LIN {X 107.589,Y -46.162,Z -55.457,A -90.000,B 90.000,C 0.000} C_DIS
LIN {X 107.509,Y -46.153,Z -55.761,A -90.000,B 90.000,C 0.000} C_DIS
LIN {X 107.348,Y -46.129,Z -56.352,A -90.000,B 90.000,C 0.000} C_DIS
LIN {X 107.212,Y -46.114,Z -56.832,A -90.000,B 90.000,C 0.000} C_DIS
LIN {X 107.081,Y -46.091,Z -57.259,A -90.000,B 90.000,C 0.000} C_DIS
LIN {X 106.960,Y -46.087,Z -57.631,A -90.000,B 90.000,C 0.000} C_DIS
LIN {X 106.873,Y -46.081,Z -57.884,A -90.000,B 90.000,C 0.000} C_DIS
LIN {X 106.583,Y -46.065,Z -58.706,A -90.000,B 90.000,C 0.000} C_DIS
LIN {X 106.300,Y -46.057,Z -59.526,A -90.000,B 90.000,C 0.000} C_DIS
LIN {X 106.266,Y -46.058,Z -59.619,A -90.000,B 90.000,C 0.000} C_DIS
LIN {X 106.210,Y -46.061,Z -59.764,A -90.000,B 90.000,C 0.000} C_DIS
LIN {X 105.890,Y -46.060,Z -60.546,A -90.000,B 90.000,C 0.000} C_DIS
LIN {X 105.587,Y -46.066,Z -61.296,A -90.000,B 90.000,C 0.000} C_DIS
LIN {X 105.326,Y -46.072,Z -61.938,A -90.000,B 90.000,C 0.000} C_DIS
LIN {X 105.166,Y -46.078,Z -62.307,A -90.000,B 90.000,C 0.000} C_DIS
LIN {X 104.885,Y -46.086,Z -62.880,A -90.000,B 90.000,C 0.000} C_DIS
LIN {X 104.370,Y -46.110,Z -63.945,A -90.000,B 90.000,C 0.000} C_DIS
LIN {X 104.116,Y -46.117,Z -64.480,A -90.000,B 90.000,C 0.000} C_DIS
LIN {X 104.061,Y -46.121,Z -64.587,A -90.000,B 90.000,C 0.000} C_DIS
LIN {X 103.858,Y -46.124,Z -64.941,A -90.000,B 90.000,C 0.000} C_DIS
LIN {X 103.565,Y -46.141,Z -65.429,A -90.000,B 90.000,C 0.000} C_DIS
LIN {X 102.922,Y -46.183,Z -66.506,A -90.000,B 90.000,C 0.000} C_DIS
LIN {X 102.789,Y -46.189,Z -66.734,A -90.000,B 90.000,C 0.000} C_DIS
LIN {X 102.578,Y -46.188,Z -67.081,A -90.000,B 90.000,C 0.000} C_DIS
LIN {X 102.463,Y -46.188,Z -67.247,A -90.000,B 90.000,C 0.000} C_DIS
LIN {X 102.227,Y -46.200,Z -67.560,A -90.000,B 90.000,C 0.000} C_DIS
LIN {X 101.675,Y -46.239,Z -68.268,A -90.000,B 90.000,C 0.000} C_DIS
LIN {X 101.476,Y -46.259,Z -68.509,A -90.000,B 90.000,C 0.000} C_DIS
LIN {X 101.020,Y -46.294,Z -69.044,A -90.000,B 90.000,C 0.000} C_DIS
LIN {X 100.781,Y -46.305,Z -69.318,A -90.000,B 90.000,C 0.000} C_DIS
LIN {X 100.500,Y -46.311,Z -69.634,A -90.000,B 90.000,C 0.000} C_DIS
LIN {X 100.413,Y -46.315,Z -69.726,A -90.000,B 90.000,C 0.000} C_DIS
LIN {X 100.368,Y -46.319,Z -69.770,A -90.000,B 90.000,C 0.000} C_DIS
LIN {X 100.015,Y -46.339,Z -70.076,A -90.000,B 90.000,C 0.000} C_DIS
LIN {X 99.523,Y -46.377,Z -70.476,A -90.000,B 90.000,C 0.000} C_DIS
LIN {X 98.816,Y -46.424,Z -71.045,A -90.000,B 90.000,C 0.000} C_DIS
LIN {X 98.553,Y -46.429,Z -71.249,A -90.000,B 90.000,C 0.000} C_DIS
LIN {X 97.950,Y -46.427,Z -71.707,A -90.000,B 90.000,C 0.000} C_DIS
LIN {X 97.860,Y -46.428,Z -71.773,A -90.000,B 90.000,C 0.000} C_DIS
LIN {X 97.743,Y -46.434,Z -71.848,A -90.000,B 90.000,C 0.000} C_DIS
LIN {X 97.472,Y -46.450,Z -72.014,A -90.000,B 90.000,C 0.000} C_DIS
LIN {X 97.222,Y -46.468,Z -72.161,A -90.000,B 90.000,C 0.000} C_DIS
LIN {X 97.080,Y -46.480,Z -72.238,A -90.000,B 90.000,C 0.000} C_DIS
LIN {X 96.822,Y -46.489,Z -72.366,A -90.000,B 90.000,C 0.000} C_DIS
LIN {X 96.112,Y -46.501,Z -72.711,A -90.000,B 90.000,C 0.000} C_DIS
LIN {X 95.963,Y -46.506,Z -72.774,A -90.000,B 90.000,C 0.000} C_DIS
LIN {X 95.665,Y -46.507,Z -72.890,A -90.000,B 90.000,C 0.000} C_DIS
LIN {X 95.513,Y -46.511,Z -72.938,A -90.000,B 90.000,C 0.000} C_DIS
LIN {X 94.694,Y -46.547,Z -73.167,A -90.000,B 90.000,C 0.000} C_DIS
LIN {X 94.626,Y -46.549,Z -73.189,A -90.000,B 90.000,C 0.000} C_DIS
LIN {X 94.421,Y -46.549,Z -73.252,A -90.000,B 90.000,C 0.000} C_DIS
LIN {X 94.032,Y -46.560,Z -73.343,A -90.000,B 90.000,C 0.000} C_DIS
LIN {X 93.943,Y -46.563,Z -73.362,A -90.000,B 90.000,C 0.000} C_DIS
LIN {X 93.880,Y -46.566,Z -73.372,A -90.000,B 90.000,C 0.000} C_DIS
LIN {X 93.755,Y -46.574,Z -73.389,A -90.000,B 90.000,C 0.000} C_DIS
LIN {X 93.477,Y -46.578,Z -73.425,A -90.000,B 90.000,C 0.000} C_DIS
LIN {X 92.687,Y -46.571,Z -73.521,A -90.000,B 90.000,C 0.000} C_DIS
LIN {X 92.591,Y -46.573,Z -73.532,A -90.000,B 90.000,C 0.000} C_DIS
LIN {X 92.407,Y -46.579,Z -73.545,A -90.000,B 90.000,C 0.000} C_DIS
LIN {X 92.089,Y -46.581,Z -73.541,A -90.000,B 90.000,C 0.000} C_DIS
LIN {X 92.022,Y -46.582,Z -73.539,A -90.000,B 90.000,C 0.000} C_DIS
LIN {X 91.526,Y -46.592,Z -73.502,A -90.000,B 90.000,C 0.000} C_DIS
LIN {X 91.111,Y -46.595,Z -73.489,A -90.000,B 90.000,C 0.000} C_DIS
LIN {X 91.023,Y -46.591,Z -73.484,A -90.000,B 90.000,C 0.000} C_DIS
LIN {X 90.905,Y -46.587,Z -73.475,A -90.000,B 90.000,C 0.000} C_DIS
LIN {X 90.779,Y -46.586,Z -73.457,A -90.000,B 90.000,C 0.000} C_DIS
LIN {X 90.544,Y -46.586,Z -73.417,A -90.000,B 90.000,C 0.000} C_DIS
LIN {X 90.416,Y -46.588,Z -73.388,A -90.000,B 90.000,C 0.000} C_DIS
LIN {X 90.003,Y -46.595,Z -73.288,A -90.000,B 90.000,C 0.000} C_DIS
LIN {X 89.846,Y -46.594,Z -73.260,A -90.000,B 90.000,C 0.000} C_DIS
LIN {X 89.559,Y -46.578,Z -73.201,A -90.000,B 90.000,C 0.000} C_DIS
LIN {X 89.440,Y -46.573,Z -73.172,A -90.000,B 90.000,C 0.000} C_DIS
LIN {X 89.132,Y -46.563,Z -73.088,A -90.000,B 90.000,C 0.000} C_DIS
LIN {X 89.029,Y -46.561,Z -73.057,A -90.000,B 90.000,C 0.000} C_DIS
LIN {X 88.840,Y -46.562,Z -72.987,A -90.000,B 90.000,C 0.000} C_DIS
LIN {X 88.626,Y -46.563,Z -72.902,A -90.000,B 90.000,C 0.000} C_DIS
LIN {X 88.200,Y -46.542,Z -72.723,A -90.000,B 90.000,C 0.000} C_DIS
LIN {X 87.848,Y -46.530,Z -72.563,A -90.000,B 90.000,C 0.000} C_DIS
LIN {X 87.511,Y -46.517,Z -72.389,A -90.000,B 90.000,C 0.000} C_DIS
LIN {X 87.327,Y -46.505,Z -72.292,A -90.000,B 90.000,C 0.000} C_DIS
LIN {X 87.280,Y -46.500,Z -72.274,A -90.000,B 90.000,C 0.000} C_DIS
LIN {X 87.174,Y -46.490,Z -72.230,A -90.000,B 90.000,C 0.000} C_DIS
LIN {X 87.006,Y -46.476,Z -72.150,A -90.000,B 90.000,C 0.000} C_DIS
LIN {X 86.828,Y -46.472,Z -72.071,A -90.000,B 90.000,C 0.000} C_DIS
LIN {X 86.767,Y -46.472,Z -72.041,A -90.000,B 90.000,C 0.000} C_DIS
LIN {X 86.689,Y -46.469,Z -71.999,A -90.000,B 90.000,C 0.000} C_DIS
LIN {X 86.578,Y -46.468,Z -71.932,A -90.000,B 90.000,C 0.000} C_DIS
LIN {X 86.493,Y -46.468,Z -71.878,A -90.000,B 90.000,C 0.000} C_DIS
LIN {X 86.279,Y -46.453,Z -71.731,A -90.000,B 90.000,C 0.000} C_DIS
LIN {X 85.850,Y -46.419,Z -71.423,A -90.000,B 90.000,C 0.000} C_DIS
LIN {X 85.760,Y -46.408,Z -71.369,A -90.000,B 90.000,C 0.000} C_DIS
LIN {X 85.585,Y -46.403,Z -71.258,A -90.000,B 90.000,C 0.000} C_DIS
LIN {X 85.416,Y -46.390,Z -71.143,A -90.000,B 90.000,C 0.000} C_DIS
LIN {X 85.343,Y -46.385,Z -71.090,A -90.000,B 90.000,C 0.000} C_DIS
LIN {X 85.266,Y -46.378,Z -71.028,A -90.000,B 90.000,C 0.000} C_DIS
LIN {X 85.091,Y -46.365,Z -70.871,A -90.000,B 90.000,C 0.000} C_DIS
LIN {X 85.014,Y -46.355,Z -70.797,A -90.000,B 90.000,C 0.000} C_DIS
LIN {X 84.936,Y -46.346,Z -70.718,A -90.000,B 90.000,C 0.000} C_DIS
LIN {X 84.756,Y -46.327,Z -70.529,A -90.000,B 90.000,C 0.000} C_DIS
LIN {X 84.658,Y -46.327,Z -70.434,A -90.000,B 90.000,C 0.000} C_DIS
LIN {X 84.355,Y -46.303,Z -70.183,A -90.000,B 90.000,C 0.000} C_DIS
LIN {X 84.253,Y -46.288,Z -70.085,A -90.000,B 90.000,C 0.000} C_DIS
LIN {X 84.127,Y -46.274,Z -69.947,A -90.000,B 90.000,C 0.000} C_DIS
LIN {X 83.956,Y -46.242,Z -69.742,A -90.000,B 90.000,C 0.000} C_DIS
LIN {X 83.874,Y -46.226,Z -69.634,A -90.000,B 90.000,C 0.000} C_DIS
LIN {X 83.782,Y -46.213,Z -69.499,A -90.000,B 90.000,C 0.000} C_DIS
LIN {X 83.711,Y -46.202,Z -69.388,A -90.000,B 90.000,C 0.000} C_DIS
LIN {X 83.619,Y -46.198,Z -69.257,A -90.000,B 90.000,C 0.000} C_DIS
LIN {X 83.569,Y -46.197,Z -69.184,A -90.000,B 90.000,C 0.000} C_DIS
LIN {X 83.433,Y -46.199,Z -68.968,A -90.000,B 90.000,C 0.000} C_DIS
LIN {X 83.314,Y -46.181,Z -68.793,A -90.000,B 90.000,C 0.000} C_DIS
LIN {X 83.245,Y -46.172,Z -68.688,A -90.000,B 90.000,C 0.000} C_DIS
LIN {X 83.110,Y -46.136,Z -68.456,A -90.000,B 90.000,C 0.000} C_DIS
LIN {X 82.973,Y -46.109,Z -68.193,A -90.000,B 90.000,C 0.000} C_DIS
LIN {X 82.834,Y -46.065,Z -67.863,A -90.000,B 90.000,C 0.000} C_DIS
LIN {X 82.812,Y -46.055,Z -67.802,A -90.000,B 90.000,C 0.000} C_DIS
LIN {X 82.777,Y -46.044,Z -67.715,A -90.000,B 90.000,C 0.000} C_DIS
LIN {X 82.723,Y -46.031,Z -67.563,A -90.000,B 90.000,C 0.000} C_DIS
LIN {X 82.697,Y -46.027,Z -67.483,A -90.000,B 90.000,C 0.000} C_DIS
LIN {X 82.592,Y -46.003,Z -67.135,A -90.000,B 90.000,C 0.000} C_DIS
LIN {X 82.505,Y -45.973,Z -66.741,A -90.000,B 90.000,C 0.000} C_DIS
LIN {X 82.442,Y -45.940,Z -66.413,A -90.000,B 90.000,C 0.000} C_DIS
LIN {X 82.413,Y -45.927,Z -66.257,A -90.000,B 90.000,C 0.000} C_DIS
LIN {X 82.375,Y -45.874,Z -65.905,A -90.000,B 90.000,C 0.000} C_DIS
LIN {X 82.362,Y -45.850,Z -65.730,A -90.000,B 90.000,C 0.000} C_DIS
LIN {X 82.347,Y -45.818,Z -65.409,A -90.000,B 90.000,C 0.000} C_DIS
LIN {X 82.364,Y -45.773,Z -65.034,A -90.000,B 90.000,C 0.000} C_DIS
LIN {X 82.401,Y -45.734,Z -64.565,A -90.000,B 90.000,C 0.000} C_DIS
LIN {X 82.410,Y -45.729,Z -64.470,A -90.000,B 90.000,C 0.000} C_DIS
LIN {X 82.479,Y -45.709,Z -63.856,A -90.000,B 90.000,C 0.000} C_DIS
LIN {X 82.501,Y -45.701,Z -63.740,A -90.000,B 90.000,C 0.000} C_DIS
LIN {X 82.576,Y -45.681,Z -63.378,A -90.000,B 90.000,C 0.000} C_DIS
LIN {X 82.598,Y -45.674,Z -63.301,A -90.000,B 90.000,C 0.000} C_DIS
LIN {X 82.709,Y -45.640,Z -62.934,A -90.000,B 90.000,C 0.000} C_DIS
LIN {X 82.820,Y -45.612,Z -62.579,A -90.000,B 90.000,C 0.000} C_DIS
LIN {X 83.043,Y -45.545,Z -62.002,A -90.000,B 90.000,C 0.000} C_DIS
LIN {X 83.069,Y -45.539,Z -61.937,A -90.000,B 90.000,C 0.000} C_DIS
LIN {X 83.136,Y -45.526,Z -61.772,A -90.000,B 90.000,C 0.000} C_DIS
LIN {X 83.311,Y -45.490,Z -61.398,A -90.000,B 90.000,C 0.000} C_DIS
LIN {X 83.482,Y -45.470,Z -61.064,A -90.000,B 90.000,C 0.000} C_DIS
LIN {X 83.601,Y -45.459,Z -60.837,A -90.000,B 90.000,C 0.000} C_DIS
LIN {X 83.737,Y -45.451,Z -60.585,A -90.000,B 90.000,C 0.000} C_DIS
LIN {X 83.897,Y -45.437,Z -60.318,A -90.000,B 90.000,C 0.000} C_DIS
LIN {X 84.064,Y -45.422,Z -60.072,A -90.000,B 90.000,C 0.000} C_DIS
LIN {X 84.175,Y -45.411,Z -59.915,A -90.000,B 90.000,C 0.000} C_DIS
LIN {X 84.538,Y -45.384,Z -59.413,A -90.000,B 90.000,C 0.000} C_DIS
LIN {X 84.832,Y -45.368,Z -59.006,A -90.000,B 90.000,C 0.000} C_DIS
LIN {X 85.043,Y -45.360,Z -58.718,A -90.000,B 90.000,C 0.000} C_DIS
LIN {X 85.401,Y -45.345,Z -58.270,A -90.000,B 90.000,C 0.000} C_DIS
LIN {X 85.618,Y -45.344,Z -57.999,A -90.000,B 90.000,C 0.000} C_DIS
LIN {X 85.618,Y -60.000,Z -57.999,A -90.000,B 90.000,C 0.000} C_DIS
LIN {X 100.781,Y -60.000,Z -71.645,A -90.000,B 90.000,C 0.000} C_DIS
LIN {X 100.781,Y -45.308,Z -71.645,A -90.000,B 90.000,C 0.000} C_DIS
LIN {X 100.498,Y -45.352,Z -71.891,A -90.000,B 90.000,C 0.000} C_DIS
LIN {X 99.019,Y -45.480,Z -73.108,A -90.000,B 90.000,C 0.000} C_DIS
LIN {X 98.875,Y -45.494,Z -73.221,A -90.000,B 90.000,C 0.000} C_DIS
LIN {X 98.794,Y -45.505,Z -73.281,A -90.000,B 90.000,C 0.000} C_DIS
LIN {X 98.634,Y -45.528,Z -73.392,A -90.000,B 90.000,C 0.000} C_DIS
LIN {X 98.370,Y -45.563,Z -73.566,A -90.000,B 90.000,C 0.000} C_DIS
LIN {X 98.120,Y -45.588,Z -73.717,A -90.000,B 90.000,C 0.000} C_DIS
LIN {X 98.017,Y -45.597,Z -73.776,A -90.000,B 90.000,C 0.000} C_DIS
LIN {X 97.761,Y -45.622,Z -73.915,A -90.000,B 90.000,C 0.000} C_DIS
LIN {X 97.649,Y -45.634,Z -73.975,A -90.000,B 90.000,C 0.000} C_DIS
LIN {X 96.893,Y -45.663,Z -74.350,A -90.000,B 90.000,C 0.000} C_DIS
LIN {X 96.728,Y -45.672,Z -74.425,A -90.000,B 90.000,C 0.000} C_DIS
LIN {X 96.420,Y -45.692,Z -74.556,A -90.000,B 90.000,C 0.000} C_DIS
LIN {X 96.325,Y -45.699,Z -74.596,A -90.000,B 90.000,C 0.000} C_DIS
LIN {X 96.224,Y -45.707,Z -74.635,A -90.000,B 90.000,C 0.000} C_DIS
LIN {X 96.046,Y -45.723,Z -74.697,A -90.000,B 90.000,C 0.000} C_DIS
LIN {X 95.705,Y -45.761,Z -74.804,A -90.000,B 90.000,C 0.000} C_DIS
LIN {X 95.483,Y -45.787,Z -74.873,A -90.000,B 90.000,C 0.000} C_DIS
LIN {X 95.195,Y -45.803,Z -74.955,A -90.000,B 90.000,C 0.000} C_DIS
LIN {X 94.962,Y -45.812,Z -75.030,A -90.000,B 90.000,C 0.000} C_DIS
LIN {X 94.827,Y -45.815,Z -75.067,A -90.000,B 90.000,C 0.000} C_DIS
LIN {X 94.711,Y -45.820,Z -75.095,A -90.000,B 90.000,C 0.000} C_DIS
LIN {X 94.438,Y -45.824,Z -75.158,A -90.000,B 90.000,C 0.000} C_DIS
LIN {X 94.221,Y -45.829,Z -75.201,A -90.000,B 90.000,C 0.000} C_DIS
LIN {X 94.075,Y -45.834,Z -75.223,A -90.000,B 90.000,C 0.000} C_DIS
LIN {X 93.969,Y -45.840,Z -75.237,A -90.000,B 90.000,C 0.000} C_DIS
LIN {X 93.730,Y -45.850,Z -75.271,A -90.000,B 90.000,C 0.000} C_DIS
LIN {X 93.009,Y -45.890,Z -75.375,A -90.000,B 90.000,C 0.000} C_DIS
LIN {X 92.771,Y -45.893,Z -75.405,A -90.000,B 90.000,C 0.000} C_DIS
LIN {X 92.521,Y -45.901,Z -75.423,A -90.000,B 90.000,C 0.000} C_DIS
LIN {X 92.379,Y -45.901,Z -75.426,A -90.000,B 90.000,C 0.000} C_DIS
LIN {X 91.977,Y -45.908,Z -75.421,A -90.000,B 90.000,C 0.000} C_DIS
LIN {X 91.870,Y -45.912,Z -75.417,A -90.000,B 90.000,C 0.000} C_DIS
LIN {X 91.504,Y -45.928,Z -75.393,A -90.000,B 90.000,C 0.000} C_DIS
LIN {X 91.385,Y -45.930,Z -75.386,A -90.000,B 90.000,C 0.000} C_DIS
LIN {X 91.019,Y -45.933,Z -75.374,A -90.000,B 90.000,C 0.000} C_DIS
LIN {X 90.836,Y -45.929,Z -75.363,A -90.000,B 90.000,C 0.000} C_DIS
LIN {X 90.711,Y -45.927,Z -75.353,A -90.000,B 90.000,C 0.000} C_DIS
LIN {X 90.460,Y -45.928,Z -75.319,A -90.000,B 90.000,C 0.000} C_DIS
LIN {X 90.240,Y -45.931,Z -75.282,A -90.000,B 90.000,C 0.000} C_DIS
LIN {X 90.113,Y -45.931,Z -75.257,A -90.000,B 90.000,C 0.000} C_DIS
LIN {X 89.726,Y -45.935,Z -75.165,A -90.000,B 90.000,C 0.000} C_DIS
LIN {X 89.607,Y -45.936,Z -75.136,A -90.000,B 90.000,C 0.000} C_DIS
LIN {X 89.499,Y -45.934,Z -75.115,A -90.000,B 90.000,C 0.000} C_DIS
LIN {X 89.141,Y -45.920,Z -75.043,A -90.000,B 90.000,C 0.000} C_DIS
LIN {X 88.963,Y -45.915,Z -74.999,A -90.000,B 90.000,C 0.000} C_DIS
LIN {X 88.762,Y -45.907,Z -74.944,A -90.000,B 90.000,C 0.000} C_DIS
LIN {X 88.540,Y -45.895,Z -74.879,A -90.000,B 90.000,C 0.000} C_DIS
LIN {X 88.439,Y -45.890,Z -74.847,A -90.000,B 90.000,C 0.000} C_DIS
LIN {X 88.145,Y -45.882,Z -74.735,A -90.000,B 90.000,C 0.000} C_DIS
LIN {X 87.825,Y -45.870,Z -74.603,A -90.000,B 90.000,C 0.000} C_DIS
LIN {X 87.611,Y -45.858,Z -74.512,A -90.000,B 90.000,C 0.000} C_DIS
LIN {X 87.445,Y -45.843,Z -74.438,A -90.000,B 90.000,C 0.000} C_DIS
LIN {X 87.096,Y -45.814,Z -74.272,A -90.000,B 90.000,C 0.000} C_DIS
LIN {X 87.015,Y -45.808,Z -74.232,A -90.000,B 90.000,C 0.000} C_DIS
LIN {X 86.829,Y -45.795,Z -74.133,A -90.000,B 90.000,C 0.000} C_DIS
LIN {X 86.590,Y -45.769,Z -74.003,A -90.000,B 90.000,C 0.000} C_DIS
LIN {X 86.455,Y -45.748,Z -73.942,A -90.000,B 90.000,C 0.000} C_DIS
LIN {X 86.043,Y -45.688,Z -73.735,A -90.000,B 90.000,C 0.000} C_DIS
LIN {X 85.980,Y -45.679,Z -73.701,A -90.000,B 90.000,C 0.000} C_DIS
LIN {X 85.792,Y -45.669,Z -73.598,A -90.000,B 90.000,C 0.000} C_DIS
LIN {X 85.536,Y -45.649,Z -73.431,A -90.000,B 90.000,C 0.000} C_DIS
LIN {X 85.302,Y -45.614,Z -73.261,A -90.000,B 90.000,C 0.000} C_DIS
LIN {X 84.913,Y -45.545,Z -72.963,A -90.000,B 90.000,C 0.000} C_DIS
LIN {X 84.803,Y -45.523,Z -72.886,A -90.000,B 90.000,C 0.000} C_DIS
LIN {X 84.696,Y -45.512,Z -72.814,A -90.000,B 90.000,C 0.000} C_DIS
LIN {X 84.404,Y -45.469,Z -72.602,A -90.000,B 90.000,C 0.000} C_DIS
LIN {X 84.281,Y -45.446,Z -72.502,A -90.000,B 90.000,C 0.000} C_DIS
LIN {X 84.167,Y -45.427,Z -72.402,A -90.000,B 90.000,C 0.000} C_DIS
LIN {X 83.903,Y -45.359,Z -72.129,A -90.000,B 90.000,C 0.000} C_DIS
LIN {X 83.784,Y -45.330,Z -71.999,A -90.000,B 90.000,C 0.000} C_DIS
LIN {X 83.595,Y -45.309,Z -71.802,A -90.000,B 90.000,C 0.000} C_DIS
LIN {X 83.587,Y -45.308,Z -71.793,A -90.000,B 90.000,C 0.000} C_DIS
LIN {X 83.467,Y -45.299,Z -71.665,A -90.000,B 90.000,C 0.000} C_DIS
LIN {X 83.253,Y -45.266,Z -71.427,A -90.000,B 90.000,C 0.000} C_DIS
LIN {X 83.072,Y -45.239,Z -71.215,A -90.000,B 90.000,C 0.000} C_DIS
LIN {X 82.923,Y -45.215,Z -71.028,A -90.000,B 90.000,C 0.000} C_DIS
LIN {X 82.861,Y -45.203,Z -70.944,A -90.000,B 90.000,C 0.000} C_DIS
LIN {X 82.758,Y -45.181,Z -70.793,A -90.000,B 90.000,C 0.000} C_DIS
LIN {X 82.718,Y -45.170,Z -70.726,A -90.000,B 90.000,C 0.000} C_DIS
LIN {X 82.658,Y -45.150,Z -70.610,A -90.000,B 90.000,C 0.000} C_DIS
LIN {X 82.632,Y -45.136,Z -70.537,A -90.000,B 90.000,C 0.000} C_DIS
LIN {X 82.621,Y -45.123,Z -70.476,A -90.000,B 90.000,C 0.000} C_DIS
LIN {X 82.620,Y -45.124,Z -70.458,A -90.000,B 90.000,C 0.000} C_DIS
LIN {X 82.624,Y -45.138,Z -70.426,A -90.000,B 90.000,C 0.000} C_DIS
LIN {X 82.634,Y -45.155,Z -70.400,A -90.000,B 90.000,C 0.000} C_DIS
LIN {X 82.650,Y -45.175,Z -70.378,A -90.000,B 90.000,C 0.000} C_DIS
LIN {X 82.685,Y -45.209,Z -70.355,A -90.000,B 90.000,C 0.000} C_DIS
LIN {X 82.716,Y -45.235,Z -70.346,A -90.000,B 90.000,C 0.000} C_DIS
LIN {X 82.752,Y -45.263,Z -70.341,A -90.000,B 90.000,C 0.000} C_DIS
LIN {X 82.794,Y -45.294,Z -70.341,A -90.000,B 90.000,C 0.000} C_DIS
LIN {X 82.841,Y -45.327,Z -70.345,A -90.000,B 90.000,C 0.000} C_DIS
LIN {X 82.950,Y -45.398,Z -70.366,A -90.000,B 90.000,C 0.000} C_DIS
LIN {X 83.080,Y -45.476,Z -70.404,A -90.000,B 90.000,C 0.000} C_DIS
LIN {X 83.227,Y -45.559,Z -70.458,A -90.000,B 90.000,C 0.000} C_DIS
LIN {X 83.392,Y -45.647,Z -70.527,A -90.000,B 90.000,C 0.000} C_DIS
LIN {X 83.573,Y -45.734,Z -70.610,A -90.000,B 90.000,C 0.000} C_DIS
LIN {X 83.669,Y -45.774,Z -70.657,A -90.000,B 90.000,C 0.000} C_DIS
LIN {X 83.768,Y -45.812,Z -70.707,A -90.000,B 90.000,C 0.000} C_DIS
LIN {X 83.871,Y -45.848,Z -70.761,A -90.000,B 90.000,C 0.000} C_DIS
LIN {X 83.978,Y -45.880,Z -70.817,A -90.000,B 90.000,C 0.000} C_DIS
LIN {X 84.316,Y -45.969,Z -71.005,A -90.000,B 90.000,C 0.000} C_DIS
LIN {X 84.555,Y -46.032,Z -71.144,A -90.000,B 90.000,C 0.000} C_DIS
LIN {X 84.804,Y -46.095,Z -71.293,A -90.000,B 90.000,C 0.000} C_DIS
LIN {X 85.061,Y -46.149,Z -71.452,A -90.000,B 90.000,C 0.000} C_DIS
LIN {X 85.326,Y -46.179,Z -71.620,A -90.000,B 90.000,C 0.000} C_DIS
LIN {X 85.598,Y -46.208,Z -71.796,A -90.000,B 90.000,C 0.000} C_DIS
LIN {X 86.155,Y -46.262,Z -72.169,A -90.000,B 90.000,C 0.000} C_DIS
LIN {X 86.439,Y -46.272,Z -72.364,A -90.000,B 90.000,C 0.000} C_DIS
LIN {X 86.725,Y -46.273,Z -72.565,A -90.000,B 90.000,C 0.000} C_DIS
LIN {X 87.011,Y -46.272,Z -72.769,A -90.000,B 90.000,C 0.000} C_DIS
LIN {X 87.296,Y -46.274,Z -72.978,A -90.000,B 90.000,C 0.000} C_DIS
LIN {X 87.580,Y -46.270,Z -73.189,A -90.000,B 90.000,C 0.000} C_DIS
LIN {X 87.862,Y -46.252,Z -73.402,A -90.000,B 90.000,C 0.000} C_DIS
LIN {X 88.411,Y -46.208,Z -73.831,A -90.000,B 90.000,C 0.000} C_DIS
LIN {X 88.808,Y -46.166,Z -74.153,A -90.000,B 90.000,C 0.000} C_DIS
LIN {X 89.062,Y -46.127,Z -74.366,A -90.000,B 90.000,C 0.000} C_DIS
LIN {X 89.308,Y -46.086,Z -74.577,A -90.000,B 90.000,C 0.000} C_DIS
LIN {X 89.656,Y -46.022,Z -74.888,A -90.000,B 90.000,C 0.000} C_DIS
LIN {X 89.874,Y -45.972,Z -75.091,A -90.000,B 90.000,C 0.000} C_DIS
LIN {X 90.079,Y -45.922,Z -75.288,A -90.000,B 90.000,C 0.000} C_DIS
LIN {X 90.269,Y -45.869,Z -75.481,A -90.000,B 90.000,C 0.000} C_DIS
LIN {X 90.444,Y -45.816,Z -75.667,A -90.000,B 90.000,C 0.000} C_DIS
LIN {X 90.603,Y -45.764,Z -75.846,A -90.000,B 90.000,C 0.000} C_DIS
LIN {X 90.743,Y -45.712,Z -76.017,A -90.000,B 90.000,C 0.000} C_DIS
LIN {X 90.807,Y -45.685,Z -76.100,A -90.000,B 90.000,C 0.000} C_DIS
LIN {X 90.919,Y -45.631,Z -76.258,A -90.000,B 90.000,C 0.000} C_DIS
LIN {X 91.011,Y -45.580,Z -76.407,A -90.000,B 90.000,C 0.000} C_DIS
LIN {X 91.081,Y -45.532,Z -76.545,A -90.000,B 90.000,C 0.000} C_DIS
LIN {X 91.118,Y -45.499,Z -76.642,A -90.000,B 90.000,C 0.000} C_DIS
LIN {X 91.142,Y -45.468,Z -76.732,A -90.000,B 90.000,C 0.000} C_DIS
LIN {X 91.151,Y -45.449,Z -76.788,A -90.000,B 90.000,C 0.000} C_DIS
LIN {X 91.153,Y -45.431,Z -76.841,A -90.000,B 90.000,C 0.000} C_DIS
LIN {X 91.144,Y -45.405,Z -76.915,A -90.000,B 90.000,C 0.000} C_DIS
LIN {X 91.130,Y -45.390,Z -76.959,A -90.000,B 90.000,C 0.000} C_DIS
LIN {X 91.109,Y -45.375,Z -77.001,A -90.000,B 90.000,C 0.000} C_DIS
LIN {X 91.065,Y -45.357,Z -77.056,A -90.000,B 90.000,C 0.000} C_DIS
LIN {X 91.005,Y -45.341,Z -77.103,A -90.000,B 90.000,C 0.000} C_DIS
LIN {X 90.955,Y -45.332,Z -77.129,A -90.000,B 90.000,C 0.000} C_DIS
LIN {X 90.898,Y -45.324,Z -77.152,A -90.000,B 90.000,C 0.000} C_DIS
LIN {X 90.834,Y -45.318,Z -77.170,A -90.000,B 90.000,C 0.000} C_DIS
LIN {X 90.762,Y -45.313,Z -77.185,A -90.000,B 90.000,C 0.000} C_DIS
LIN {X 90.681,Y -45.310,Z -77.195,A -90.000,B 90.000,C 0.000} C_DIS
LIN {X 90.593,Y -45.308,Z -77.200,A -90.000,B 90.000,C 0.000} C_DIS
LIN {X 90.497,Y -45.307,Z -77.202,A -90.000,B 90.000,C 0.000} C_DIS
LIN {X 90.336,Y -45.308,Z -77.195,A -90.000,B 90.000,C 0.000} C_DIS
LIN {X 90.218,Y -45.310,Z -77.185,A -90.000,B 90.000,C 0.000} C_DIS
LIN {X 90.092,Y -45.312,Z -77.170,A -90.000,B 90.000,C 0.000} C_DIS
LIN {X 89.957,Y -45.312,Z -77.151,A -90.000,B 90.000,C 0.000} C_DIS
LIN {X 89.659,Y -45.310,Z -77.096,A -90.000,B 90.000,C 0.000} C_DIS
LIN {X 89.497,Y -45.311,Z -77.062,A -90.000,B 90.000,C 0.000} C_DIS
LIN {X 89.324,Y -45.308,Z -77.022,A -90.000,B 90.000,C 0.000} C_DIS
LIN {X 89.209,Y -45.310,Z -76.994,A -90.000,B 90.000,C 0.000} C_DIS
LIN {X 89.143,Y -45.308,Z -76.981,A -90.000,B 90.000,C 0.000} C_DIS
LIN {X 89.143,Y -60.000,Z -76.981,A -90.000,B 90.000,C 0.000} C_DIS
LIN {X 105.925,Y -60.000,Z -41.896,A -90.000,B 90.000,C 0.000} C_DIS
LIN {X 105.925,Y -45.308,Z -41.896,A -90.000,B 90.000,C 0.000} C_DIS
LIN {X 106.082,Y -45.344,Z -41.934,A -90.000,B 90.000,C 0.000} C_DIS
LIN {X 106.366,Y -45.411,Z -42.013,A -90.000,B 90.000,C 0.000} C_DIS
LIN {X 106.501,Y -45.443,Z -42.052,A -90.000,B 90.000,C 0.000} C_DIS
LIN {X 106.671,Y -45.474,Z -42.117,A -90.000,B 90.000,C 0.000} C_DIS
LIN {X 106.787,Y -45.496,Z -42.167,A -90.000,B 90.000,C 0.000} C_DIS
LIN {X 107.089,Y -45.544,Z -42.310,A -90.000,B 90.000,C 0.000} C_DIS
LIN {X 107.241,Y -45.573,Z -42.387,A -90.000,B 90.000,C 0.000} C_DIS
LIN {X 107.476,Y -45.607,Z -42.514,A -90.000,B 90.000,C 0.000} C_DIS
LIN {X 107.642,Y -45.623,Z -42.620,A -90.000,B 90.000,C 0.000} C_DIS
LIN {X 107.730,Y -45.632,Z -42.680,A -90.000,B 90.000,C 0.000} C_DIS
LIN {X 107.976,Y -45.648,Z -42.875,A -90.000,B 90.000,C 0.000} C_DIS
LIN {X 108.217,Y -45.649,Z -43.084,A -90.000,B 90.000,C 0.000} C_DIS
LIN {X 108.349,Y -45.643,Z -43.218,A -90.000,B 90.000,C 0.000} C_DIS
LIN {X 108.438,Y -45.640,Z -43.312,A -90.000,B 90.000,C 0.000} C_DIS
LIN {X 108.637,Y -45.621,Z -43.557,A -90.000,B 90.000,C 0.000} C_DIS
LIN {X 108.696,Y -45.609,Z -43.634,A -90.000,B 90.000,C 0.000} C_DIS
LIN {X 108.801,Y -45.598,Z -43.769,A -90.000,B 90.000,C 0.000} C_DIS
LIN {X 108.914,Y -45.579,Z -43.938,A -90.000,B 90.000,C 0.000} C_DIS
LIN {X 108.962,Y -45.572,Z -44.012,A -90.000,B 90.000,C 0.000} C_DIS
LIN {X 109.100,Y -45.534,Z -44.270,A -90.000,B 90.000,C 0.000} C_DIS
LIN {X 109.231,Y -45.483,Z -44.539,A -90.000,B 90.000,C 0.000} C_DIS
LIN {X 109.265,Y -45.467,Z -44.621,A -90.000,B 90.000,C 0.000} C_DIS
LIN {X 109.337,Y -45.433,Z -44.804,A -90.000,B 90.000,C 0.000} C_DIS
LIN {X 109.416,Y -45.380,Z -45.063,A -90.000,B 90.000,C 0.000} C_DIS
LIN {X 109.495,Y -45.308,Z -45.369,A -90.000,B 90.000,C 0.000} C_DIS
LIN {X 109.495,Y -45.308,Z -45.370,A -90.000,B 90.000,C 0.000} C_DIS
LIN {X 109.488,Y -45.308,Z -45.439,A -90.000,B 90.000,C 0.000} C_DIS
LIN {X 109.447,Y -45.308,Z -45.810,A -90.000,B 90.000,C 0.000} C_DIS
LIN {X 109.401,Y -45.308,Z -46.112,A -90.000,B 90.000,C 0.000} C_DIS
LIN {X 109.374,Y -45.308,Z -46.271,A -90.000,B 90.000,C 0.000} C_DIS
LIN {X 109.322,Y -45.308,Z -46.535,A -90.000,B 90.000,C 0.000} C_DIS
LIN {X 109.233,Y -45.308,Z -47.115,A -90.000,B 90.000,C 0.000} C_DIS
LIN {X 109.262,Y -45.308,Z -47.223,A -90.000,B 90.000,C 0.000} C_DIS
LIN {X 109.319,Y -45.308,Z -47.388,A -90.000,B 90.000,C 0.000} C_DIS
LIN {X 109.423,Y -45.308,Z -47.744,A -90.000,B 90.000,C 0.000} C_DIS
LIN {X 109.517,Y -45.308,Z -48.133,A -90.000,B 90.000,C 0.000} C_DIS
LIN {X 109.629,Y -45.308,Z -48.632,A -90.000,B 90.000,C 0.000} C_DIS
LIN {X 109.704,Y -45.308,Z -48.975,A -90.000,B 90.000,C 0.000} C_DIS
LIN {X 109.717,Y -45.308,Z -49.043,A -90.000,B 90.000,C 0.000} C_DIS
LIN {X 109.742,Y -45.308,Z -49.394,A -90.000,B 90.000,C 0.000} C_DIS
LIN {X 109.749,Y -45.308,Z -49.650,A -90.000,B 90.000,C 0.000} C_DIS
LIN {X 109.743,Y -45.308,Z -50.059,A -90.000,B 90.000,C 0.000} C_DIS
LIN {X 109.740,Y -45.308,Z -50.164,A -90.000,B 90.000,C 0.000} C_DIS
LIN {X 109.698,Y -45.308,Z -50.955,A -90.000,B 90.000,C 0.000} C_DIS
LIN {X 109.641,Y -45.308,Z -51.330,A -90.000,B 90.000,C 0.000} C_DIS
LIN {X 109.545,Y -45.308,Z -51.893,A -90.000,B 90.000,C 0.000} C_DIS
LIN {X 109.498,Y -45.308,Z -52.109,A -90.000,B 90.000,C 0.000} C_DIS
LIN {X 109.239,Y -45.308,Z -53.232,A -90.000,B 90.000,C 0.000} C_DIS
LIN {X 109.133,Y -45.308,Z -53.621,A -90.000,B 90.000,C 0.000} C_DIS
LIN {X 109.006,Y -45.308,Z -54.037,A -90.000,B 90.000,C 0.000} C_DIS
LIN {X 108.942,Y -45.308,Z -54.229,A -90.000,B 90.000,C 0.000} C_DIS
LIN {X 108.596,Y -45.308,Z -55.236,A -90.000,B 90.000,C 0.000} C_DIS
LIN {X 108.299,Y -45.308,Z -56.144,A -90.000,B 90.000,C 0.000} C_DIS
LIN {X 107.704,Y -45.308,Z -57.852,A -90.000,B 90.000,C 0.000} C_DIS
LIN {X 106.964,Y -45.308,Z -59.825,A -90.000,B 90.000,C 0.000} C_DIS
LIN {X 106.812,Y -45.308,Z -60.255,A -90.000,B 90.000,C 0.000} C_DIS
LIN {X 106.144,Y -45.308,Z -61.954,A -90.000,B 90.000,C 0.000} C_DIS
LIN {X 105.967,Y -45.308,Z -62.424,A -90.000,B 90.000,C 0.000} C_DIS
LIN {X 105.044,Y -45.308,Z -64.560,A -90.000,B 90.000,C 0.000} C_DIS
LIN {X 105.005,Y -45.308,Z -64.654,A -90.000,B 90.000,C 0.000} C_DIS
LIN {X 104.830,Y -45.308,Z -65.024,A -90.000,B 90.000,C 0.000} C_DIS
LIN {X 103.931,Y -45.308,Z -66.836,A -90.000,B 90.000,C 0.000} C_DIS
LIN {X 103.799,Y -45.308,Z -67.116,A -90.000,B 90.000,C 0.000} C_DIS
LIN {X 103.631,Y -45.308,Z -67.412,A -90.000,B 90.000,C 0.000} C_DIS
LIN {X 103.092,Y -45.308,Z -68.340,A -90.000,B 90.000,C 0.000} C_DIS
LIN {X 102.260,Y -45.308,Z -69.683,A -90.000,B 90.000,C 0.000} C_DIS
LIN {X 101.871,Y -45.308,Z -70.240,A -90.000,B 90.000,C 0.000} C_DIS
LIN {X 100.896,Y -45.308,Z -71.498,A -90.000,B 90.000,C 0.000} C_DIS
LIN {X 100.560,Y -45.308,Z -71.923,A -90.000,B 90.000,C 0.000} C_DIS
LIN {X 100.323,Y -45.308,Z -72.162,A -90.000,B 90.000,C 0.000} C_DIS
LIN {X 98.829,Y -45.308,Z -73.723,A -90.000,B 90.000,C 0.000} C_DIS
LIN {X 98.575,Y -45.308,Z -73.966,A -90.000,B 90.000,C 0.000} C_DIS
LIN {X 97.874,Y -45.308,Z -74.566,A -90.000,B 90.000,C 0.000} C_DIS
LIN {X 97.002,Y -45.308,Z -75.243,A -90.000,B 90.000,C 0.000} C_DIS
LIN {X 96.664,Y -45.308,Z -75.446,A -90.000,B 90.000,C 0.000} C_DIS
LIN {X 96.388,Y -45.308,Z -75.607,A -90.000,B 90.000,C 0.000} C_DIS
LIN {X 94.627,Y -45.308,Z -76.482,A -90.000,B 90.000,C 0.000} C_DIS
LIN {X 94.370,Y -45.308,Z -76.590,A -90.000,B 90.000,C 0.000} C_DIS
LIN {X 94.208,Y -45.308,Z -76.653,A -90.000,B 90.000,C 0.000} C_DIS
LIN {X 94.110,Y -45.308,Z -76.689,A -90.000,B 90.000,C 0.000} C_DIS
LIN {X 93.807,Y -45.308,Z -76.796,A -90.000,B 90.000,C 0.000} C_DIS
LIN {X 92.749,Y -45.308,Z -77.004,A -90.000,B 90.000,C 0.000} C_DIS
LIN {X 92.087,Y -45.308,Z -77.142,A -90.000,B 90.000,C 0.000} C_DIS
LIN {X 91.809,Y -45.308,Z -77.188,A -90.000,B 90.000,C 0.000} C_DIS
LIN {X 91.691,Y -45.308,Z -77.195,A -90.000,B 90.000,C 0.000} C_DIS
LIN {X 91.430,Y -45.308,Z -77.193,A -90.000,B 90.000,C 0.000} C_DIS
LIN {X 90.720,Y -45.308,Z -77.194,A -90.000,B 90.000,C 0.000} C_DIS
LIN {X 90.128,Y -45.308,Z -77.182,A -90.000,B 90.000,C 0.000} C_DIS
LIN {X 89.942,Y -45.308,Z -77.145,A -90.000,B 90.000,C 0.000} C_DIS
LIN {X 89.220,Y -45.308,Z -77.001,A -90.000,B 90.000,C 0.000} C_DIS
LIN {X 88.694,Y -45.308,Z -76.868,A -90.000,B 90.000,C 0.000} C_DIS
LIN {X 88.431,Y -45.308,Z -76.766,A -90.000,B 90.000,C 0.000} C_DIS
LIN {X 88.041,Y -45.308,Z -76.591,A -90.000,B 90.000,C 0.000} C_DIS
LIN {X 87.462,Y -45.308,Z -76.268,A -90.000,B 90.000,C 0.000} C_DIS
LIN {X 87.222,Y -45.308,Z -76.121,A -90.000,B 90.000,C 0.000} C_DIS
LIN {X 86.909,Y -45.308,Z -75.893,A -90.000,B 90.000,C 0.000} C_DIS
LIN {X 86.698,Y -45.308,Z -75.706,A -90.000,B 90.000,C 0.000} C_DIS
LIN {X 86.176,Y -45.308,Z -75.219,A -90.000,B 90.000,C 0.000} C_DIS
LIN {X 85.841,Y -45.308,Z -74.816,A -90.000,B 90.000,C 0.000} C_DIS
LIN {X 85.769,Y -45.308,Z -74.715,A -90.000,B 90.000,C 0.000} C_DIS
LIN {X 85.256,Y -45.308,Z -74.210,A -90.000,B 90.000,C 0.000} C_DIS
LIN {X 85.052,Y -45.308,Z -73.964,A -90.000,B 90.000,C 0.000} C_DIS
LIN {X 84.908,Y -45.308,Z -73.721,A -90.000,B 90.000,C 0.000} C_DIS
LIN {X 84.407,Y -45.308,Z -73.061,A -90.000,B 90.000,C 0.000} C_DIS
LIN {X 84.289,Y -45.308,Z -72.926,A -90.000,B 90.000,C 0.000} C_DIS
LIN {X 84.086,Y -45.308,Z -72.645,A -90.000,B 90.000,C 0.000} C_DIS
LIN {X 83.761,Y -45.308,Z -72.027,A -90.000,B 90.000,C 0.000} C_DIS
LIN {X 83.685,Y -45.308,Z -71.928,A -90.000,B 90.000,C 0.000} C_DIS
LIN {X 83.479,Y -45.308,Z -71.643,A -90.000,B 90.000,C 0.000} C_DIS
LIN {X 83.295,Y -45.308,Z -71.343,A -90.000,B 90.000,C 0.000} C_DIS
LIN {X 83.119,Y -45.308,Z -71.008,A -90.000,B 90.000,C 0.000} C_DIS
LIN {X 83.007,Y -45.308,Z -70.706,A -90.000,B 90.000,C 0.000} C_DIS
LIN {X 82.660,Y -45.308,Z -70.016,A -90.000,B 90.000,C 0.000} C_DIS
LIN {X 82.617,Y -45.308,Z -69.919,A -90.000,B 90.000,C 0.000} C_DIS
LIN {X 82.424,Y -45.308,Z -69.420,A -90.000,B 90.000,C 0.000} C_DIS
LIN {X 82.317,Y -45.308,Z -69.031,A -90.000,B 90.000,C 0.000} C_DIS
LIN {X 82.236,Y -45.308,Z -68.616,A -90.000,B 90.000,C 0.000} C_DIS
LIN {X 82.180,Y -45.308,Z -68.314,A -90.000,B 90.000,C 0.000} C_DIS
LIN {X 82.122,Y -45.308,Z -68.102,A -90.000,B 90.000,C 0.000} C_DIS
LIN {X 81.991,Y -45.308,Z -67.526,A -90.000,B 90.000,C 0.000} C_DIS
LIN {X 81.956,Y -45.308,Z -67.196,A -90.000,B 90.000,C 0.000} C_DIS
LIN {X 81.912,Y -45.308,Z -66.724,A -90.000,B 90.000,C 0.000} C_DIS
LIN {X 81.914,Y -45.308,Z -66.583,A -90.000,B 90.000,C 0.000} C_DIS
LIN {X 81.927,Y -45.308,Z -66.099,A -90.000,B 90.000,C 0.000} C_DIS
LIN {X 82.108,Y -45.308,Z -64.721,A -90.000,B 90.000,C 0.000} C_DIS
LIN {X 82.162,Y -45.308,Z -64.369,A -90.000,B 90.000,C 0.000} C_DIS
LIN {X 82.364,Y -45.308,Z -63.452,A -90.000,B 90.000,C 0.000} C_DIS
LIN {X 82.505,Y -45.308,Z -63.007,A -90.000,B 90.000,C 0.000} C_DIS
LIN {X 82.909,Y -45.308,Z -62.079,A -90.000,B 90.000,C 0.000} C_DIS
LIN {X 83.123,Y -45.308,Z -61.654,A -90.000,B 90.000,C 0.000} C_DIS
LIN {X 83.357,Y -45.308,Z -61.210,A -90.000,B 90.000,C 0.000} C_DIS
LIN {X 83.589,Y -45.308,Z -60.786,A -90.000,B 90.000,C 0.000} C_DIS
LIN {X 83.894,Y -45.308,Z -60.285,A -90.000,B 90.000,C 0.000} C_DIS
LIN {X 83.997,Y -45.308,Z -60.137,A -90.000,B 90.000,C 0.000} C_DIS
LIN {X 84.175,Y -45.308,Z -59.890,A -90.000,B 90.000,C 0.000} C_DIS
LIN {X 84.969,Y -45.308,Z -58.805,A -90.000,B 90.000,C 0.000} C_DIS
LIN {X 85.606,Y -45.308,Z -58.010,A -90.000,B 90.000,C 0.000} C_DIS
LIN {X 85.729,Y -45.308,Z -57.860,A -90.000,B 90.000,C 0.000} C_DIS
LIN {X 85.730,Y -45.308,Z -57.859,A -90.000,B 90.000,C 0.000} C_DIS
LIN {X 86.058,Y -45.308,Z -57.495,A -90.000,B 90.000,C 0.000} C_DIS
LIN {X 87.795,Y -45.308,Z -55.685,A -90.000,B 90.000,C 0.000} C_DIS
LIN {X 89.687,Y -45.308,Z -53.953,A -90.000,B 90.000,C 0.000} C_DIS
LIN {X 90.146,Y -45.308,Z -53.537,A -90.000,B 90.000,C 0.000} C_DIS
LIN {X 92.218,Y -45.308,Z -51.761,A -90.000,B 90.000,C 0.000} C_DIS
LIN {X 94.367,Y -45.308,Z -49.945,A -90.000,B 90.000,C 0.000} C_DIS
LIN {X 96.069,Y -45.308,Z -48.454,A -90.000,B 90.000,C 0.000} C_DIS
LIN {X 96.319,Y -45.308,Z -48.211,A -90.000,B 90.000,C 0.000} C_DIS
LIN {X 97.421,Y -45.308,Z -47.177,A -90.000,B 90.000,C 0.000} C_DIS
LIN {X 97.804,Y -45.308,Z -46.825,A -90.000,B 90.000,C 0.000} C_DIS
LIN {X 97.880,Y -45.308,Z -46.758,A -90.000,B 90.000,C 0.000} C_DIS
LIN {X 98.685,Y -45.308,Z -46.007,A -90.000,B 90.000,C 0.000} C_DIS
LIN {X 99.460,Y -45.308,Z -45.342,A -90.000,B 90.000,C 0.000} C_DIS
LIN {X 99.831,Y -45.308,Z -45.037,A -90.000,B 90.000,C 0.000} C_DIS
LIN {X 100.481,Y -45.308,Z -44.518,A -90.000,B 90.000,C 0.000} C_DIS
LIN {X 100.641,Y -45.308,Z -44.404,A -90.000,B 90.000,C 0.000} C_DIS
LIN {X 101.429,Y -45.308,Z -43.841,A -90.000,B 90.000,C 0.000} C_DIS
LIN {X 101.813,Y -45.308,Z -43.596,A -90.000,B 90.000,C 0.000} C_DIS
LIN {X 102.100,Y -45.308,Z -43.426,A -90.000,B 90.000,C 0.000} C_DIS
LIN {X 102.765,Y -45.308,Z -43.037,A -90.000,B 90.000,C 0.000} C_DIS
LIN {X 102.958,Y -45.308,Z -42.935,A -90.000,B 90.000,C 0.000} C_DIS
LIN {X 103.755,Y -45.308,Z -42.549,A -90.000,B 90.000,C 0.000} C_DIS
LIN {X 104.149,Y -45.308,Z -42.393,A -90.000,B 90.000,C 0.000} C_DIS
LIN {X 104.859,Y -45.308,Z -42.134,A -90.000,B 90.000,C 0.000} C_DIS
LIN {X 105.484,Y -45.308,Z -41.980,A -90.000,B 90.000,C 0.000} C_DIS
LIN {X 105.760,Y -45.308,Z -41.922,A -90.000,B 90.000,C 0.000} C_DIS
LIN {X 105.855,Y -45.308,Z -41.901,A -90.000,B 90.000,C 0.000} C_DIS
LIN {X 106.361,Y -45.308,Z -41.859,A -90.000,B 90.000,C 0.000} C_DIS
LIN {X 106.712,Y -45.308,Z -41.836,A -90.000,B 90.000,C 0.000} C_DIS
LIN {X 107.062,Y -45.308,Z -41.863,A -90.000,B 90.000,C 0.000} C_DIS
LIN {X 107.199,Y -45.308,Z -41.888,A -90.000,B 90.000,C 0.000} C_DIS
LIN {X 107.308,Y -45.308,Z -41.897,A -90.000,B 90.000,C 0.000} C_DIS
LIN {X 107.660,Y -45.308,Z -41.939,A -90.000,B 90.000,C 0.000} C_DIS
LIN {X 107.970,Y -45.308,Z -42.015,A -90.000,B 90.000,C 0.000} C_DIS
LIN {X 108.265,Y -45.308,Z -42.139,A -90.000,B 90.000,C 0.000} C_DIS
LIN {X 108.536,Y -45.308,Z -42.307,A -90.000,B 90.000,C 0.000} C_DIS
LIN {X 108.778,Y -45.308,Z -42.515,A -90.000,B 90.000,C 0.000} C_DIS
LIN {X 108.985,Y -45.308,Z -42.759,A -90.000,B 90.000,C 0.000} C_DIS
LIN {X 109.025,Y -45.308,Z -42.824,A -90.000,B 90.000,C 0.000} C_DIS
LIN {X 109.171,Y -45.308,Z -43.028,A -90.000,B 90.000,C 0.000} C_DIS
LIN {X 109.295,Y -45.308,Z -43.250,A -90.000,B 90.000,C 0.000} C_DIS
LIN {X 109.416,Y -45.308,Z -43.545,A -90.000,B 90.000,C 0.000} C_DIS
LIN {X 109.491,Y -45.308,Z -43.856,A -90.000,B 90.000,C 0.000} C_DIS
LIN {X 109.508,Y -45.308,Z -44.076,A -90.000,B 90.000,C 0.000} C_DIS
LIN {X 109.518,Y -45.308,Z -44.228,A -90.000,B 90.000,C 0.000} C_DIS
LIN {X 109.544,Y -45.308,Z -44.584,A -90.000,B 90.000,C 0.000} C_DIS
LIN {X 109.532,Y -45.308,Z -44.985,A -90.000,B 90.000,C 0.000} C_DIS
LIN {X 109.495,Y -45.308,Z -45.370,A -90.000,B 90.000,C 0.000} C_DIS
LIN {X 109.495,Y -60.000,Z -45.370,A -90.000,B 90.000,C 0.000} C_DIS
LIN {X 96.327,Y -60.000,Z -48.204,A -90.000,B 90.000,C 0.000} C_DIS
LIN {X 96.327,Y -43.308,Z -48.204,A -90.000,B 90.000,C 0.000} C_DIS
LIN {X 97.663,Y -43.309,Z -46.906,A -90.000,B 90.000,C 0.000} C_DIS
LIN {X 98.608,Y -43.312,Z -45.908,A -90.000,B 90.000,C 0.000} C_DIS
LIN {X 99.094,Y -43.318,Z -45.395,A -90.000,B 90.000,C 0.000} C_DIS
LIN {X 99.470,Y -43.328,Z -44.976,A -90.000,B 90.000,C 0.000} C_DIS
LIN {X 99.964,Y -43.347,Z -44.428,A -90.000,B 90.000,C 0.000} C_DIS
LIN {X 100.289,Y -43.363,Z -44.083,A -90.000,B 90.000,C 0.000} C_DIS
LIN {X 100.587,Y -43.386,Z -43.765,A -90.000,B 90.000,C 0.000} C_DIS
LIN {X 100.913,Y -43.405,Z -43.455,A -90.000,B 90.000,C 0.000} C_DIS
LIN {X 101.192,Y -43.426,Z -43.190,A -90.000,B 90.000,C 0.000} C_DIS
LIN {X 101.442,Y -43.449,Z -42.958,A -90.000,B 90.000,C 0.000} C_DIS
LIN {X 101.501,Y -43.456,Z -42.904,A -90.000,B 90.000,C 0.000} C_DIS
LIN {X 101.860,Y -43.490,Z -42.602,A -90.000,B 90.000,C 0.000} C_DIS
LIN {X 102.069,Y -43.509,Z -42.433,A -90.000,B 90.000,C 0.000} C_DIS
LIN {X 102.339,Y -43.533,Z -42.221,A -90.000,B 90.000,C 0.000} C_DIS
LIN {X 102.421,Y -43.541,Z -42.159,A -90.000,B 90.000,C 0.000} C_DIS
LIN {X 102.583,Y -43.556,Z -42.044,A -90.000,B 90.000,C 0.000} C_DIS
LIN {X 102.931,Y -43.596,Z -41.800,A -90.000,B 90.000,C 0.000} C_DIS
LIN {X 103.281,Y -43.631,Z -41.568,A -90.000,B 90.000,C 0.000} C_DIS
LIN {X 103.535,Y -43.661,Z -41.417,A -90.000,B 90.000,C 0.000} C_DIS
LIN {X 103.752,Y -43.686,Z -41.293,A -90.000,B 90.000,C 0.000} C_DIS
LIN {X 103.996,Y -43.719,Z -41.157,A -90.000,B 90.000,C 0.000} C_DIS
LIN {X 104.072,Y -43.729,Z -41.115,A -90.000,B 90.000,C 0.000} C_DIS
LIN {X 104.470,Y -43.766,Z -40.921,A -90.000,B 90.000,C 0.000} C_DIS
LIN {X 104.654,Y -43.794,Z -40.839,A -90.000,B 90.000,C 0.000} C_DIS
LIN {X 104.842,Y -43.825,Z -40.757,A -90.000,B 90.000,C 0.000} C_DIS
LIN {X 105.153,Y -43.866,Z -40.635,A -90.000,B 90.000,C 0.000} C_DIS
LIN {X 105.301,Y -43.886,Z -40.582,A -90.000,B 90.000,C 0.000} C_DIS
LIN {X 105.556,Y -43.919,Z -40.495,A -90.000,B 90.000,C 0.000} C_DIS
LIN {X 105.653,Y -43.933,Z -40.463,A -90.000,B 90.000,C 0.000} C_DIS
LIN {X 105.826,Y -43.968,Z -40.414,A -90.000,B 90.000,C 0.000} C_DIS
LIN {X 106.133,Y -44.020,Z -40.343,A -90.000,B 90.000,C 0.000} C_DIS
LIN {X 106.432,Y -44.064,Z -40.285,A -90.000,B 90.000,C 0.000} C_DIS
LIN {X 106.622,Y -44.094,Z -40.250,A -90.000,B 90.000,C 0.000} C_DIS
LIN {X 106.746,Y -44.117,Z -40.230,A -90.000,B 90.000,C 0.000} C_DIS
LIN {X 106.846,Y -44.131,Z -40.225,A -90.000,B 90.000,C 0.000} C_DIS
LIN {X 107.195,Y -44.188,Z -40.212,A -90.000,B 90.000,C 0.000} C_DIS
LIN {X 107.358,Y -44.218,Z -40.213,A -90.000,B 90.000,C 0.000} C_DIS
LIN {X 107.418,Y -44.230,Z -40.216,A -90.000,B 90.000,C 0.000} C_DIS
LIN {X 107.561,Y -44.254,Z -40.216,A -90.000,B 90.000,C 0.000} C_DIS
LIN {X 107.885,Y -44.285,Z -40.235,A -90.000,B 90.000,C 0.000} C_DIS
LIN {X 107.946,Y -44.291,Z -40.241,A -90.000,B 90.000,C 0.000} C_DIS
LIN {X 108.046,Y -44.303,Z -40.254,A -90.000,B 90.000,C 0.000} C_DIS
LIN {X 108.328,Y -44.348,Z -40.297,A -90.000,B 90.000,C 0.000} C_DIS
LIN {X 108.465,Y -44.369,Z -40.320,A -90.000,B 90.000,C 0.000} C_DIS
LIN {X 108.550,Y -44.385,Z -40.339,A -90.000,B 90.000,C 0.000} C_DIS
LIN {X 108.682,Y -44.403,Z -40.380,A -90.000,B 90.000,C 0.000} C_DIS
LIN {X 108.830,Y -44.425,Z -40.430,A -90.000,B 90.000,C 0.000} C_DIS
LIN {X 108.962,Y -44.440,Z -40.478,A -90.000,B 90.000,C 0.000} C_DIS
LIN {X 109.077,Y -44.456,Z -40.522,A -90.000,B 90.000,C 0.000} C_DIS
LIN {X 109.140,Y -44.464,Z -40.551,A -90.000,B 90.000,C 0.000} C_DIS
LIN {X 109.231,Y -44.477,Z -40.598,A -90.000,B 90.000,C 0.000} C_DIS
LIN {X 109.385,Y -44.500,Z -40.681,A -90.000,B 90.000,C 0.000} C_DIS
LIN {X 109.576,Y -44.514,Z -40.795,A -90.000,B 90.000,C 0.000} C_DIS
LIN {X 109.653,Y -44.521,Z -40.846,A -90.000,B 90.000,C 0.000} C_DIS
LIN {X 109.764,Y -44.528,Z -40.934,A -90.000,B 90.000,C 0.000} C_DIS
LIN {X 109.892,Y -44.537,Z -41.039,A -90.000,B 90.000,C 0.000} C_DIS
LIN {X 110.042,Y -44.544,Z -41.166,A -90.000,B 90.000,C 0.000} C_DIS
LIN {X 110.069,Y -44.546,Z -41.191,A -90.000,B 90.000,C 0.000} C_DIS
LIN {X 110.156,Y -44.552,Z -41.278,A -90.000,B 90.000,C 0.000} C_DIS
LIN {X 110.201,Y -44.556,Z -41.328,A -90.000,B 90.000,C 0.000} C_DIS
LIN {X 110.385,Y -44.565,Z -41.539,A -90.000,B 90.000,C 0.000} C_DIS
LIN {X 110.491,Y -44.563,Z -41.674,A -90.000,B 90.000,C 0.000} C_DIS
LIN {X 110.532,Y -44.563,Z -41.733,A -90.000,B 90.000,C 0.000} C_DIS
LIN {X 110.574,Y -44.563,Z -41.800,A -90.000,B 90.000,C 0.000} C_DIS
LIN {X 110.667,Y -44.556,Z -41.934,A -90.000,B 90.000,C 0.000} C_DIS
LIN {X 110.724,Y -44.548,Z -42.024,A -90.000,B 90.000,C 0.000} C_DIS
LIN {X 110.783,Y -44.541,Z -42.128,A -90.000,B 90.000,C 0.000} C_DIS
LIN {X 110.821,Y -44.538,Z -42.198,A -90.000,B 90.000,C 0.000} C_DIS
LIN {X 110.899,Y -44.520,Z -42.354,A -90.000,B 90.000,C 0.000} C_DIS
LIN {X 110.950,Y -44.509,Z -42.462,A -90.000,B 90.000,C 0.000} C_DIS
LIN {X 110.964,Y -44.506,Z -42.495,A -90.000,B 90.000,C 0.000} C_DIS
LIN {X 111.090,Y -44.459,Z -42.855,A -90.000,B 90.000,C 0.000} C_DIS
LIN {X 111.141,Y -44.440,Z -43.024,A -90.000,B 90.000,C 0.000} C_DIS
LIN {X 111.151,Y -44.435,Z -43.067,A -90.000,B 90.000,C 0.000} C_DIS
LIN {X 111.217,Y -44.387,Z -43.443,A -90.000,B 90.000,C 0.000} C_DIS
LIN {X 111.226,Y -44.379,Z -43.502,A -90.000,B 90.000,C 0.000} C_DIS
LIN {X 111.241,Y -44.362,Z -43.659,A -90.000,B 90.000,C 0.000} C_DIS
LIN {X 111.244,Y -44.354,Z -43.733,A -90.000,B 90.000,C 0.000} C_DIS
LIN {X 111.247,Y -44.326,Z -43.973,A -90.000,B 90.000,C 0.000} C_DIS
LIN {X 111.238,Y -44.248,Z -44.510,A -90.000,B 90.000,C 0.000} C_DIS
LIN {X 111.229,Y -44.233,Z -44.634,A -90.000,B 90.000,C 0.000} C_DIS
LIN {X 111.190,Y -44.191,Z -45.033,A -90.000,B 90.000,C 0.000} C_DIS
LIN {X 111.171,Y -44.178,Z -45.183,A -90.000,B 90.000,C 0.000} C_DIS
LIN {X 111.146,Y -44.167,Z -45.357,A -90.000,B 90.000,C 0.000} C_DIS
LIN {X 111.133,Y -44.167,Z -45.489,A -90.000,B 90.000,C 0.000} C_DIS
LIN {X 111.107,Y -44.200,Z -45.943,A -90.000,B 90.000,C 0.000} C_DIS
LIN {X 111.094,Y -44.225,Z -46.160,A -90.000,B 90.000,C 0.000} C_DIS
LIN {X 111.067,Y -44.281,Z -46.551,A -90.000,B 90.000,C 0.000} C_DIS
LIN {X 111.043,Y -44.319,Z -46.791,A -90.000,B 90.000,C 0.000} C_DIS
LIN {X 111.030,Y -44.339,Z -46.934,A -90.000,B 90.000,C 0.000} C_DIS
LIN {X 111.026,Y -44.345,Z -46.983,A -90.000,B 90.000,C 0.000} C_DIS
LIN {X 111.071,Y -44.332,Z -47.160,A -90.000,B 90.000,C 0.000} C_DIS
LIN {X 111.093,Y -44.322,Z -47.258,A -90.000,B 90.000,C 0.000} C_DIS
LIN {X 111.156,Y -44.295,Z -47.576,A -90.000,B 90.000,C 0.000} C_DIS
LIN {X 111.217,Y -44.269,Z -47.905,A -90.000,B 90.000,C 0.000} C_DIS
LIN {X 111.234,Y -44.257,Z -48.012,A -90.000,B 90.000,C 0.000} C_DIS
LIN {X 111.308,Y -44.219,Z -48.456,A -90.000,B 90.000,C 0.000} C_DIS
LIN {X 111.338,Y -44.184,Z -48.714,A -90.000,B 90.000,C 0.000} C_DIS
LIN {X 111.342,Y -44.178,Z -48.761,A -90.000,B 90.000,C 0.000} C_DIS
LIN {X 111.349,Y -44.158,Z -48.930,A -90.000,B 90.000,C 0.000} C_DIS
LIN {X 111.349,Y -44.124,Z -49.279,A -90.000,B 90.000,C 0.000} C_DIS
LIN {X 111.339,Y -44.096,Z -49.607,A -90.000,B 90.000,C 0.000} C_DIS
LIN {X 111.302,Y -44.059,Z -50.160,A -90.000,B 90.000,C 0.000} C_DIS
LIN {X 111.298,Y -44.056,Z -50.214,A -90.000,B 90.000,C 0.000} C_DIS
LIN {X 111.187,Y -43.978,Z -51.069,A -90.000,B 90.000,C 0.000} C_DIS
LIN {X 111.159,Y -43.965,Z -51.203,A -90.000,B 90.000,C 0.000} C_DIS
LIN {X 111.067,Y -43.933,Z -51.601,A -90.000,B 90.000,C 0.000} C_DIS
LIN {X 110.965,Y -43.904,Z -52.031,A -90.000,B 90.000,C 0.000} C_DIS
LIN {X 110.924,Y -43.891,Z -52.189,A -90.000,B 90.000,C 0.000} C_DIS
LIN {X 110.858,Y -43.876,Z -52.425,A -90.000,B 90.000,C 0.000} C_DIS
LIN {X 110.725,Y -43.852,Z -52.890,A -90.000,B 90.000,C 0.000} C_DIS
LIN {X 110.590,Y -43.825,Z -53.346,A -90.000,B 90.000,C 0.000} C_DIS
LIN {X 110.511,Y -43.805,Z -53.581,A -90.000,B 90.000,C 0.000} C_DIS
LIN {X 110.364,Y -43.779,Z -54.002,A -90.000,B 90.000,C 0.000} C_DIS
LIN {X 110.315,Y -43.773,Z -54.137,A -90.000,B 90.000,C 0.000} C_DIS
LIN {X 110.210,Y -43.763,Z -54.438,A -90.000,B 90.000,C 0.000} C_DIS
LIN {X 109.906,Y -43.750,Z -55.279,A -90.000,B 90.000,C 0.000} C_DIS
LIN {X 109.776,Y -43.742,Z -55.632,A -90.000,B 90.000,C 0.000} C_DIS
LIN {X 109.443,Y -43.717,Z -56.543,A -90.000,B 90.000,C 0.000} C_DIS
LIN {X 109.167,Y -43.707,Z -57.294,A -90.000,B 90.000,C 0.000} C_DIS
LIN {X 108.805,Y -43.691,Z -58.266,A -90.000,B 90.000,C 0.000} C_DIS
LIN {X 108.679,Y -43.690,Z -58.598,A -90.000,B 90.000,C 0.000} C_DIS
LIN {X 108.543,Y -43.695,Z -58.979,A -90.000,B 90.000,C 0.000} C_DIS
LIN {X 108.076,Y -43.702,Z -60.252,A -90.000,B 90.000,C 0.000} C_DIS
LIN {X 107.919,Y -43.701,Z -60.690,A -90.000,B 90.000,C 0.000} C_DIS
LIN {X 107.767,Y -43.708,Z -61.105,A -90.000,B 90.000,C 0.000} C_DIS
LIN {X 107.630,Y -43.713,Z -61.470,A -90.000,B 90.000,C 0.000} C_DIS
LIN {X 107.284,Y -43.725,Z -62.392,A -90.000,B 90.000,C 0.000} C_DIS
LIN {X 107.089,Y -43.727,Z -62.917,A -90.000,B 90.000,C 0.000} C_DIS
LIN {X 106.694,Y -43.755,Z -63.919,A -90.000,B 90.000,C 0.000} C_DIS
LIN {X 106.171,Y -43.779,Z -65.203,A -90.000,B 90.000,C 0.000} C_DIS
LIN {X 105.997,Y -43.790,Z -65.603,A -90.000,B 90.000,C 0.000} C_DIS
LIN {X 105.944,Y -43.795,Z -65.722,A -90.000,B 90.000,C 0.000} C_DIS
LIN {X 105.154,Y -43.846,Z -67.441,A -90.000,B 90.000,C 0.000} C_DIS
LIN {X 105.031,Y -43.845,Z -67.701,A -90.000,B 90.000,C 0.000} C_DIS
LIN {X 104.961,Y -43.850,Z -67.840,A -90.000,B 90.000,C 0.000} C_DIS
LIN {X 104.821,Y -43.857,Z -68.104,A -90.000,B 90.000,C 0.000} C_DIS
LIN {X 104.291,Y -43.893,Z -69.088,A -90.000,B 90.000,C 0.000} C_DIS
LIN {X 103.903,Y -43.932,Z -69.786,A -90.000,B 90.000,C 0.000} C_DIS
LIN {X 103.739,Y -43.942,Z -70.069,A -90.000,B 90.000,C 0.000} C_DIS
LIN {X 103.461,Y -43.947,Z -70.523,A -90.000,B 90.000,C 0.000} C_DIS
LIN {X 103.092,Y -43.973,Z -71.092,A -90.000,B 90.000,C 0.000} C_DIS
LIN {X 102.794,Y -44.006,Z -71.527,A -90.000,B 90.000,C 0.000} C_DIS
LIN {X 102.194,Y -44.050,Z -72.361,A -90.000,B 90.000,C 0.000} C_DIS
LIN {X 101.955,Y -44.058,Z -72.676,A -90.000,B 90.000,C 0.000} C_DIS
LIN {X 101.789,Y -44.065,Z -72.894,A -90.000,B 90.000,C 0.000} C_DIS
LIN {X 101.708,Y -44.069,Z -72.993,A -90.000,B 90.000,C 0.000} C_DIS
LIN {X 101.461,Y -44.095,Z -73.272,A -90.000,B 90.000,C 0.000} C_DIS
LIN {X 100.537,Y -44.184,Z -74.331,A -90.000,B 90.000,C 0.000} C_DIS
LIN {X 100.280,Y -44.201,Z -74.616,A -90.000,B 90.000,C 0.000} C_DIS
LIN {X 99.985,Y -44.213,Z -74.933,A -90.000,B 90.000,C 0.000} C_DIS
LIN {X 99.739,Y -44.230,Z -75.183,A -90.000,B 90.000,C 0.000} C_DIS
LIN {X 99.670,Y -44.236,Z -75.250,A -90.000,B 90.000,C 0.000} C_DIS
LIN {X 99.300,Y -44.276,Z -75.600,A -90.000,B 90.000,C 0.000} C_DIS
LIN {X 98.996,Y -44.295,Z -75.876,A -90.000,B 90.000,C 0.000} C_DIS
LIN {X 98.931,Y -44.301,Z -75.933,A -90.000,B 90.000,C 0.000} C_DIS
LIN {X 98.625,Y -44.329,Z -76.191,A -90.000,B 90.000,C 0.000} C_DIS
LIN {X 98.339,Y -44.348,Z -76.427,A -90.000,B 90.000,C 0.000} C_DIS
LIN {X 98.077,Y -44.349,Z -76.630,A -90.000,B 90.000,C 0.000} C_DIS
LIN {X 97.988,Y -44.351,Z -76.696,A -90.000,B 90.000,C 0.000} C_DIS
LIN {X 97.907,Y -44.354,Z -76.750,A -90.000,B 90.000,C 0.000} C_DIS
LIN {X 97.518,Y -44.378,Z -76.998,A -90.000,B 90.000,C 0.000} C_DIS
LIN {X 97.285,Y -44.392,Z -77.142,A -90.000,B 90.000,C 0.000} C_DIS
LIN {X 97.181,Y -44.399,Z -77.203,A -90.000,B 90.000,C 0.000} C_DIS
LIN {X 96.392,Y -44.469,Z -77.632,A -90.000,B 90.000,C 0.000} C_DIS
LIN {X 95.508,Y -44.517,Z -78.095,A -90.000,B 90.000,C 0.000} C_DIS
LIN {X 95.367,Y -44.522,Z -78.166,A -90.000,B 90.000,C 0.000} C_DIS
LIN {X 95.254,Y -44.529,Z -78.217,A -90.000,B 90.000,C 0.000} C_DIS
LIN {X 95.026,Y -44.530,Z -78.311,A -90.000,B 90.000,C 0.000} C_DIS
LIN {X 94.835,Y -44.532,Z -78.386,A -90.000,B 90.000,C 0.000} C_DIS
LIN {X 94.423,Y -44.540,Z -78.537,A -90.000,B 90.000,C 0.000} C_DIS
LIN {X 94.299,Y -44.544,Z -78.578,A -90.000,B 90.000,C 0.000} C_DIS
LIN {X 94.130,Y -44.553,Z -78.620,A -90.000,B 90.000,C 0.000} C_DIS
LIN {X 93.670,Y -44.581,Z -78.722,A -90.000,B 90.000,C 0.000} C_DIS
LIN {X 93.116,Y -44.609,Z -78.841,A -90.000,B 90.000,C 0.000} C_DIS
LIN {X 92.684,Y -44.623,Z -78.937,A -90.000,B 90.000,C 0.000} C_DIS
LIN {X 92.399,Y -44.620,Z -78.994,A -90.000,B 90.000,C 0.000} C_DIS
LIN {X 92.052,Y -44.618,Z -79.049,A -90.000,B 90.000,C 0.000} C_DIS
LIN {X 91.876,Y -44.622,Z -79.066,A -90.000,B 90.000,C 0.000} C_DIS
LIN {X 91.817,Y -44.623,Z -79.070,A -90.000,B 90.000,C 0.000} C_DIS
LIN {X 91.671,Y -44.629,Z -79.076,A -90.000,B 90.000,C 0.000} C_DIS
LIN {X 91.236,Y -44.650,Z -79.082,A -90.000,B 90.000,C 0.000} C_DIS
LIN {X 90.857,Y -44.665,Z -79.087,A -90.000,B 90.000,C 0.000} C_DIS
LIN {X 90.574,Y -44.664,Z -79.085,A -90.000,B 90.000,C 0.000} C_DIS
LIN {X 90.090,Y -44.662,Z -79.074,A -90.000,B 90.000,C 0.000} C_DIS
LIN {X 89.983,Y -44.663,Z -79.069,A -90.000,B 90.000,C 0.000} C_DIS
LIN {X 89.855,Y -44.666,Z -79.056,A -90.000,B 90.000,C 0.000} C_DIS
LIN {X 89.751,Y -44.670,Z -79.039,A -90.000,B 90.000,C 0.000} C_DIS
LIN {X 89.300,Y -44.696,Z -78.958,A -90.000,B 90.000,C 0.000} C_DIS
LIN {X 89.024,Y -44.696,Z -78.903,A -90.000,B 90.000,C 0.000} C_DIS
LIN {X 88.822,Y -44.693,Z -78.862,A -90.000,B 90.000,C 0.000} C_DIS
LIN {X 88.206,Y -44.693,Z -78.707,A -90.000,B 90.000,C 0.000} C_DIS
LIN {X 88.137,Y -44.693,Z -78.688,A -90.000,B 90.000,C 0.000} C_DIS
LIN {X 87.998,Y -44.697,Z -78.641,A -90.000,B 90.000,C 0.000} C_DIS
LIN {X 87.943,Y -44.699,Z -78.620,A -90.000,B 90.000,C 0.000} C_DIS
LIN {X 87.680,Y -44.699,Z -78.517,A -90.000,B 90.000,C 0.000} C_DIS
LIN {X 87.345,Y -44.689,Z -78.363,A -90.000,B 90.000,C 0.000} C_DIS
LIN {X 87.263,Y -44.686,Z -78.325,A -90.000,B 90.000,C 0.000} C_DIS
LIN {X 87.173,Y -44.683,Z -78.281,A -90.000,B 90.000,C 0.000} C_DIS
LIN {X 86.520,Y -44.670,Z -77.913,A -90.000,B 90.000,C 0.000} C_DIS
LIN {X 86.238,Y -44.650,Z -77.733,A -90.000,B 90.000,C 0.000} C_DIS
LIN {X 86.158,Y -44.644,Z -77.679,A -90.000,B 90.000,C 0.000} C_DIS
LIN {X 86.104,Y -44.641,Z -77.639,A -90.000,B 90.000,C 0.000} C_DIS
LIN {X 85.803,Y -44.610,Z -77.406,A -90.000,B 90.000,C 0.000} C_DIS
LIN {X 85.693,Y -44.601,Z -77.314,A -90.000,B 90.000,C 0.000} C_DIS
LIN {X 85.427,Y -44.582,Z -77.069,A -90.000,B 90.000,C 0.000} C_DIS
LIN {X 85.134,Y -44.562,Z -76.784,A -90.000,B 90.000,C 0.000} C_DIS
LIN {X 84.920,Y -44.528,Z -76.566,A -90.000,B 90.000,C 0.000} C_DIS
LIN {X 84.829,Y -44.510,Z -76.463,A -90.000,B 90.000,C 0.000} C_DIS
LIN {X 84.736,Y -44.496,Z -76.346,A -90.000,B 90.000,C 0.000} C_DIS
LIN {X 84.406,Y -44.485,Z -75.940,A -90.000,B 90.000,C 0.000} C_DIS
LIN {X 84.379,Y -44.483,Z -75.903,A -90.000,B 90.000,C 0.000} C_DIS
LIN {X 84.231,Y -44.459,Z -75.742,A -90.000,B 90.000,C 0.000} C_DIS
LIN {X 83.961,Y -44.407,Z -75.439,A -90.000,B 90.000,C 0.000} C_DIS
LIN {X 83.932,Y -44.402,Z -75.404,A -90.000,B 90.000,C 0.000} C_DIS
LIN {X 83.866,Y -44.381,Z -75.310,A -90.000,B 90.000,C 0.000} C_DIS
LIN {X 83.697,Y -44.357,Z -75.085,A -90.000,B 90.000,C 0.000} C_DIS
LIN {X 83.565,Y -44.344,Z -74.891,A -90.000,B 90.000,C 0.000} C_DIS
LIN {X 83.472,Y -44.340,Z -74.730,A -90.000,B 90.000,C 0.000} C_DIS
LIN {X 83.447,Y -44.340,Z -74.691,A -90.000,B 90.000,C 0.000} C_DIS
LIN {X 83.272,Y -44.317,Z -74.438,A -90.000,B 90.000,C 0.000} C_DIS
LIN {X 83.077,Y -44.278,Z -74.144,A -90.000,B 90.000,C 0.000} C_DIS
LIN {X 83.056,Y -44.274,Z -74.116,A -90.000,B 90.000,C 0.000} C_DIS
LIN {X 82.978,Y -44.248,Z -74.001,A -90.000,B 90.000,C 0.000} C_DIS
LIN {X 82.896,Y -44.225,Z -73.868,A -90.000,B 90.000,C 0.000} C_DIS
LIN {X 82.740,Y -44.183,Z -73.606,A -90.000,B 90.000,C 0.000} C_DIS
LIN {X 82.682,Y -44.180,Z -73.514,A -90.000,B 90.000,C 0.000} C_DIS
LIN {X 82.619,Y -44.179,Z -73.401,A -90.000,B 90.000,C 0.000} C_DIS
LIN {X 82.470,Y -44.179,Z -73.119,A -90.000,B 90.000,C 0.000} C_DIS
LIN {X 82.373,Y -44.165,Z -72.914,A -90.000,B 90.000,C 0.000} C_DIS
LIN {X 82.152,Y -44.108,Z -72.537,A -90.000,B 90.000,C 0.000} C_DIS
LIN {X 82.054,Y -44.071,Z -72.326,A -90.000,B 90.000,C 0.000} C_DIS
LIN {X 82.037,Y -44.064,Z -72.287,A -90.000,B 90.000,C 0.000} C_DIS
LIN {X 81.969,Y -44.050,Z -72.153,A -90.000,B 90.000,C 0.000} C_DIS
LIN {X 81.925,Y -44.042,Z -72.063,A -90.000,B 90.000,C 0.000} C_DIS
LIN {X 81.762,Y -44.017,Z -71.709,A -90.000,B 90.000,C 0.000} C_DIS
LIN {X 81.679,Y -44.013,Z -71.508,A -90.000,B 90.000,C 0.000} C_DIS
LIN {X 81.614,Y -44.005,Z -71.312,A -90.000,B 90.000,C 0.000} C_DIS
LIN {X 81.471,Y -43.966,Z -70.953,A -90.000,B 90.000,C 0.000} C_DIS
LIN {X 81.352,Y -43.919,Z -70.617,A -90.000,B 90.000,C 0.000} C_DIS
LIN {X 81.298,Y -43.890,Z -70.420,A -90.000,B 90.000,C 0.000} C_DIS
LIN {X 81.197,Y -43.843,Z -70.020,A -90.000,B 90.000,C 0.000} C_DIS
LIN {X 81.143,Y -43.829,Z -69.832,A -90.000,B 90.000,C 0.000} C_DIS
LIN {X 81.094,Y -43.824,Z -69.636,A -90.000,B 90.000,C 0.000} C_DIS
LIN {X 81.038,Y -43.812,Z -69.385,A -90.000,B 90.000,C 0.000} C_DIS
LIN {X 81.006,Y -43.810,Z -69.226,A -90.000,B 90.000,C 0.000} C_DIS
LIN {X 80.978,Y -43.809,Z -69.079,A -90.000,B 90.000,C 0.000} C_DIS
LIN {X 80.918,Y -43.783,Z -68.601,A -90.000,B 90.000,C 0.000} C_DIS
LIN {X 80.888,Y -43.762,Z -68.391,A -90.000,B 90.000,C 0.000} C_DIS
LIN {X 80.851,Y -43.689,Z -67.808,A -90.000,B 90.000,C 0.000} C_DIS
LIN {X 80.853,Y -43.679,Z -67.750,A -90.000,B 90.000,C 0.000} C_DIS
LIN {X 80.859,Y -43.661,Z -67.609,A -90.000,B 90.000,C 0.000} C_DIS
LIN {X 80.883,Y -43.618,Z -67.191,A -90.000,B 90.000,C 0.000} C_DIS
LIN {X 80.891,Y -43.601,Z -66.994,A -90.000,B 90.000,C 0.000} C_DIS
LIN {X 80.901,Y -43.585,Z -66.819,A -90.000,B 90.000,C 0.000} C_DIS
LIN {X 80.909,Y -43.578,Z -66.709,A -90.000,B 90.000,C 0.000} C_DIS
LIN {X 80.957,Y -43.558,Z -66.145,A -90.000,B 90.000,C 0.000} C_DIS
LIN {X 80.986,Y -43.548,Z -65.973,A -90.000,B 90.000,C 0.000} C_DIS
LIN {X 81.103,Y -43.532,Z -65.322,A -90.000,B 90.000,C 0.000} C_DIS
LIN {X 81.215,Y -43.506,Z -64.865,A -90.000,B 90.000,C 0.000} C_DIS
LIN {X 81.226,Y -43.503,Z -64.825,A -90.000,B 90.000,C 0.000} C_DIS
LIN {X 81.339,Y -43.473,Z -64.503,A -90.000,B 90.000,C 0.000} C_DIS
LIN {X 81.447,Y -43.447,Z -64.210,A -90.000,B 90.000,C 0.000} C_DIS
LIN {X 81.510,Y -43.437,Z -64.050,A -90.000,B 90.000,C 0.000} C_DIS
LIN {X 81.630,Y -43.418,Z -63.753,A -90.000,B 90.000,C 0.000} C_DIS
LIN {X 81.849,Y -43.383,Z -63.288,A -90.000,B 90.000,C 0.000} C_DIS
LIN {X 81.955,Y -43.373,Z -63.069,A -90.000,B 90.000,C 0.000} C_DIS
LIN {X 82.067,Y -43.362,Z -62.871,A -90.000,B 90.000,C 0.000} C_DIS
LIN {X 82.380,Y -43.346,Z -62.321,A -90.000,B 90.000,C 0.000} C_DIS
LIN {X 82.652,Y -43.336,Z -61.855,A -90.000,B 90.000,C 0.000} C_DIS
LIN {X 82.707,Y -43.334,Z -61.765,A -90.000,B 90.000,C 0.000} C_DIS
LIN {X 82.970,Y -43.326,Z -61.378,A -90.000,B 90.000,C 0.000} C_DIS
LIN {X 83.460,Y -43.314,Z -60.705,A -90.000,B 90.000,C 0.000} C_DIS
LIN {X 84.096,Y -43.311,Z -59.832,A -90.000,B 90.000,C 0.000} C_DIS
LIN {X 84.253,Y -43.311,Z -59.618,A -90.000,B 90.000,C 0.000} C_DIS
LIN {X 85.599,Y -43.308,Z -58.015,A -90.000,B 90.000,C 0.000} C_DIS
LIN {X 85.637,Y -43.308,Z -57.970,A -90.000,B 90.000,C 0.000} C_DIS
LIN {X 85.705,Y -43.308,Z -57.888,A -90.000,B 90.000,C 0.000} C_DIS
LIN {X 86.298,Y -43.309,Z -57.179,A -90.000,B 90.000,C 0.000} C_DIS
LIN {X 86.741,Y -43.309,Z -56.643,A -90.000,B 90.000,C 0.000} C_DIS
LIN {X 87.476,Y -43.309,Z -55.736,A -90.000,B 90.000,C 0.000} C_DIS
LIN {X 87.490,Y -43.309,Z -55.726,A -90.000,B 90.000,C 0.000} C_DIS
LIN {X 87.516,Y -43.309,Z -55.738,A -90.000,B 90.000,C 0.000} C_DIS
LIN {X 87.546,Y -43.309,Z -55.733,A -90.000,B 90.000,C 0.000} C_DIS
LIN {X 87.603,Y -43.309,Z -55.709,A -90.000,B 90.000,C 0.000} C_DIS
LIN {X 87.659,Y -43.309,Z -55.676,A -90.000,B 90.000,C 0.000} C_DIS
LIN {X 87.734,Y -43.309,Z -55.627,A -90.000,B 90.000,C 0.000} C_DIS
LIN {X 87.829,Y -43.309,Z -55.559,A -90.000,B 90.000,C 0.000} C_DIS
LIN {X 88.095,Y -43.308,Z -55.352,A -90.000,B 90.000,C 0.000} C_DIS
LIN {X 88.479,Y -43.308,Z -55.031,A -90.000,B 90.000,C 0.000} C_DIS
LIN {X 88.722,Y -43.308,Z -54.820,A -90.000,B 90.000,C 0.000} C_DIS
LIN {X 89.002,Y -43.308,Z -54.572,A -90.000,B 90.000,C 0.000} C_DIS
LIN {X 89.321,Y -43.308,Z -54.281,A -90.000,B 90.000,C 0.000} C_DIS
LIN {X 89.688,Y -43.308,Z -53.952,A -90.000,B 90.000,C 0.000} C_DIS
LIN {X 89.717,Y -43.308,Z -53.926,A -90.000,B 90.000,C 0.000} C_DIS
LIN {X 90.919,Y -43.308,Z -52.827,A -90.000,B 90.000,C 0.000} C_DIS
LIN {X 90.937,Y -43.308,Z -52.813,A -90.000,B 90.000,C 0.000} C_DIS
LIN {X 90.946,Y -43.308,Z -52.814,A -90.000,B 90.000,C 0.000} C_DIS
LIN {X 90.967,Y -43.308,Z -52.803,A -90.000,B 90.000,C 0.000} C_DIS
LIN {X 91.017,Y -43.308,Z -52.767,A -90.000,B 90.000,C 0.000} C_DIS
LIN {X 91.264,Y -43.308,Z -52.569,A -90.000,B 90.000,C 0.000} C_DIS
LIN {X 91.490,Y -43.308,Z -52.380,A -90.000,B 90.000,C 0.000} C_DIS
LIN {X 91.802,Y -43.307,Z -52.113,A -90.000,B 90.000,C 0.000} C_DIS
LIN {X 92.219,Y -43.308,Z -51.761,A -90.000,B 90.000,C 0.000} C_DIS
LIN {X 92.263,Y -43.308,Z -51.722,A -90.000,B 90.000,C 0.000} C_DIS
LIN {X 92.263,Y -60.000,Z -51.722,A -90.000,B 90.000,C 0.000} C_DIS
LIN {X 109.275,Y -60.000,Z -38.814,A -90.000,B 90.000,C 0.000} C_DIS
LIN {X 109.275,Y -43.308,Z -38.814,A -90.000,B 90.000,C 0.000} C_DIS
LIN {X 109.543,Y -43.378,Z -38.882,A -90.000,B 90.000,C 0.000} C_DIS
LIN {X 109.742,Y -43.429,Z -38.938,A -90.000,B 90.000,C 0.000} C_DIS
LIN {X 109.904,Y -43.463,Z -38.996,A -90.000,B 90.000,C 0.000} C_DIS
LIN {X 110.045,Y -43.497,Z -39.053,A -90.000,B 90.000,C 0.000} C_DIS
LIN {X 110.314,Y -43.562,Z -39.178,A -90.000,B 90.000,C 0.000} C_DIS
LIN {X 110.599,Y -43.619,Z -39.327,A -90.000,B 90.000,C 0.000} C_DIS
LIN {X 110.636,Y -43.627,Z -39.349,A -90.000,B 90.000,C 0.000} C_DIS
LIN {X 110.732,Y -43.640,Z -39.411,A -90.000,B 90.000,C 0.000} C_DIS
LIN {X 110.916,Y -43.670,Z -39.542,A -90.000,B 90.000,C 0.000} C_DIS
LIN {X 110.943,Y -43.675,Z -39.562,A -90.000,B 90.000,C 0.000} C_DIS
LIN {X 111.213,Y -43.705,Z -39.779,A -90.000,B 90.000,C 0.000} C_DIS
LIN {X 111.327,Y -43.719,Z -39.875,A -90.000,B 90.000,C 0.000} C_DIS
LIN {X 111.469,Y -43.739,Z -40.007,A -90.000,B 90.000,C 0.000} C_DIS
LIN {X 111.545,Y -43.752,Z -40.082,A -90.000,B 90.000,C 0.000} C_DIS
LIN {X 111.752,Y -43.771,Z -40.312,A -90.000,B 90.000,C 0.000} C_DIS
LIN {X 111.842,Y -43.772,Z -40.421,A -90.000,B 90.000,C 0.000} C_DIS
LIN {X 111.953,Y -43.775,Z -40.559,A -90.000,B 90.000,C 0.000} C_DIS
LIN {X 112.034,Y -43.771,Z -40.677,A -90.000,B 90.000,C 0.000} C_DIS
LIN {X 112.097,Y -43.769,Z -40.774,A -90.000,B 90.000,C 0.000} C_DIS
LIN {X 112.132,Y -43.767,Z -40.824,A -90.000,B 90.000,C 0.000} C_DIS
LIN {X 112.214,Y -43.754,Z -40.951,A -90.000,B 90.000,C 0.000} C_DIS
LIN {X 112.299,Y -43.742,Z -41.091,A -90.000,B 90.000,C 0.000} C_DIS
LIN {X 112.385,Y -43.732,Z -41.245,A -90.000,B 90.000,C 0.000} C_DIS
LIN {X 112.430,Y -43.724,Z -41.332,A -90.000,B 90.000,C 0.000} C_DIS
LIN {X 112.543,Y -43.697,Z -41.564,A -90.000,B 90.000,C 0.000} C_DIS
LIN {X 112.570,Y -43.689,Z -41.623,A -90.000,B 90.000,C 0.000} C_DIS
LIN {X 112.628,Y -43.665,Z -41.771,A -90.000,B 90.000,C 0.000} C_DIS
LIN {X 112.664,Y -43.651,Z -41.875,A -90.000,B 90.000,C 0.000} C_DIS
LIN {X 112.744,Y -43.609,Z -42.116,A -90.000,B 90.000,C 0.000} C_DIS
LIN {X 112.771,Y -43.593,Z -42.203,A -90.000,B 90.000,C 0.000} C_DIS
LIN {X 112.838,Y -43.543,Z -42.464,A -90.000,B 90.000,C 0.000} C_DIS
LIN {X 112.860,Y -43.526,Z -42.567,A -90.000,B 90.000,C 0.000} C_DIS
LIN {X 112.893,Y -43.498,Z -42.754,A -90.000,B 90.000,C 0.000} C_DIS
LIN {X 112.937,Y -43.424,Z -43.101,A -90.000,B 90.000,C 0.000} C_DIS
LIN {X 112.946,Y -43.397,Z -43.225,A -90.000,B 90.000,C 0.000} C_DIS
LIN {X 112.954,Y -43.359,Z -43.410,A -90.000,B 90.000,C 0.000} C_DIS
LIN {X 112.950,Y -43.319,Z -43.590,A -90.000,B 90.000,C 0.000} C_DIS
LIN {X 112.947,Y -43.308,Z -43.645,A -90.000,B 90.000,C 0.000} C_DIS
LIN {X 112.947,Y -60.000,Z -43.645,A -90.000,B 90.000,C 0.000} C_DIS
LIN {X 98.381,Y -60.000,Z -78.451,A -90.000,B 90.000,C 0.000} C_DIS
LIN {X 98.381,Y -43.308,Z -78.451,A -90.000,B 90.000,C 0.000} C_DIS
LIN {X 98.078,Y -43.353,Z -78.656,A -90.000,B 90.000,C 0.000} C_DIS
LIN {X 97.932,Y -43.376,Z -78.749,A -90.000,B 90.000,C 0.000} C_DIS
LIN {X 97.390,Y -43.468,Z -79.072,A -90.000,B 90.000,C 0.000} C_DIS
LIN {X 96.773,Y -43.558,Z -79.429,A -90.000,B 90.000,C 0.000} C_DIS
LIN {X 96.174,Y -43.604,Z -79.749,A -90.000,B 90.000,C 0.000} C_DIS
LIN {X 96.029,Y -43.611,Z -79.819,A -90.000,B 90.000,C 0.000} C_DIS
LIN {X 95.737,Y -43.629,Z -79.949,A -90.000,B 90.000,C 0.000} C_DIS
LIN {X 95.436,Y -43.648,Z -80.077,A -90.000,B 90.000,C 0.000} C_DIS
LIN {X 94.962,Y -43.685,Z -80.263,A -90.000,B 90.000,C 0.000} C_DIS
LIN {X 94.775,Y -43.703,Z -80.329,A -90.000,B 90.000,C 0.000} C_DIS
LIN {X 94.532,Y -43.734,Z -80.400,A -90.000,B 90.000,C 0.000} C_DIS
LIN {X 94.002,Y -43.807,Z -80.536,A -90.000,B 90.000,C 0.000} C_DIS
LIN {X 93.748,Y -43.825,Z -80.592,A -90.000,B 90.000,C 0.000} C_DIS
LIN {X 93.467,Y -43.837,Z -80.653,A -90.000,B 90.000,C 0.000} C_DIS
LIN {X 92.771,Y -43.858,Z -80.805,A -90.000,B 90.000,C 0.000} C_DIS
LIN {X 92.644,Y -43.863,Z -80.830,A -90.000,B 90.000,C 0.000} C_DIS
LIN {X 92.341,Y -43.877,Z -80.884,A -90.000,B 90.000,C 0.000} C_DIS
LIN {X 92.214,Y -43.885,Z -80.903,A -90.000,B 90.000,C 0.000} C_DIS
LIN {X 92.000,Y -43.899,Z -80.927,A -90.000,B 90.000,C 0.000} C_DIS
LIN {X 91.826,Y -43.911,Z -80.940,A -90.000,B 90.000,C 0.000} C_DIS
LIN {X 91.642,Y -43.926,Z -80.949,A -90.000,B 90.000,C 0.000} C_DIS
LIN {X 91.391,Y -43.940,Z -80.952,A -90.000,B 90.000,C 0.000} C_DIS
LIN {X 90.842,Y -43.960,Z -80.959,A -90.000,B 90.000,C 0.000} C_DIS
LIN {X 90.497,Y -43.974,Z -80.960,A -90.000,B 90.000,C 0.000} C_DIS
LIN {X 89.998,Y -43.995,Z -80.957,A -90.000,B 90.000,C 0.000} C_DIS
LIN {X 89.891,Y -43.998,Z -80.953,A -90.000,B 90.000,C 0.000} C_DIS
LIN {X 89.773,Y -44.000,Z -80.944,A -90.000,B 90.000,C 0.000} C_DIS
LIN {X 89.585,Y -44.005,Z -80.924,A -90.000,B 90.000,C 0.000} C_DIS
LIN {X 89.498,Y -44.009,Z -80.911,A -90.000,B 90.000,C 0.000} C_DIS
LIN {X 89.264,Y -44.019,Z -80.871,A -90.000,B 90.000,C 0.000} C_DIS
LIN {X 88.501,Y -44.067,Z -80.735,A -90.000,B 90.000,C 0.000} C_DIS
LIN {X 88.362,Y -44.068,Z -80.705,A -90.000,B 90.000,C 0.000} C_DIS
LIN {X 88.228,Y -44.070,Z -80.672,A -90.000,B 90.000,C 0.000} C_DIS
LIN {X 87.684,Y -44.068,Z -80.534,A -90.000,B 90.000,C 0.000} C_DIS
LIN {X 87.510,Y -44.071,Z -80.482,A -90.000,B 90.000,C 0.000} C_DIS
LIN {X 87.281,Y -44.078,Z -80.403,A -90.000,B 90.000,C 0.000} C_DIS
LIN {X 87.170,Y -44.081,Z -80.360,A -90.000,B 90.000,C 0.000} C_DIS
LIN {X 86.950,Y -44.081,Z -80.273,A -90.000,B 90.000,C 0.000} C_DIS
LIN {X 86.526,Y -44.061,Z -80.077,A -90.000,B 90.000,C 0.000} C_DIS
LIN {X 86.351,Y -44.051,Z -79.991,A -90.000,B 90.000,C 0.000} C_DIS
LIN {X 86.258,Y -44.047,Z -79.941,A -90.000,B 90.000,C 0.000} C_DIS
LIN {X 85.811,Y -44.029,Z -79.686,A -90.000,B 90.000,C 0.000} C_DIS
LIN {X 85.606,Y -44.013,Z -79.566,A -90.000,B 90.000,C 0.000} C_DIS
LIN {X 85.529,Y -44.002,Z -79.516,A -90.000,B 90.000,C 0.000} C_DIS
LIN {X 85.223,Y -43.955,Z -79.310,A -90.000,B 90.000,C 0.000} C_DIS
LIN {X 85.079,Y -43.934,Z -79.206,A -90.000,B 90.000,C 0.000} C_DIS
LIN {X 84.984,Y -43.921,Z -79.133,A -90.000,B 90.000,C 0.000} C_DIS
LIN {X 84.653,Y -43.871,Z -78.866,A -90.000,B 90.000,C 0.000} C_DIS
LIN {X 84.544,Y -43.856,Z -78.772,A -90.000,B 90.000,C 0.000} C_DIS
LIN {X 84.467,Y -43.847,Z -78.703,A -90.000,B 90.000,C 0.000} C_DIS
LIN {X 84.274,Y -43.814,Z -78.515,A -90.000,B 90.000,C 0.000} C_DIS
LIN {X 84.165,Y -43.783,Z -78.398,A -90.000,B 90.000,C 0.000} C_DIS
LIN {X 83.986,Y -43.734,Z -78.203,A -90.000,B 90.000,C 0.000} C_DIS
LIN {X 83.759,Y -43.665,Z -77.949,A -90.000,B 90.000,C 0.000} C_DIS
LIN {X 83.600,Y -43.635,Z -77.778,A -90.000,B 90.000,C 0.000} C_DIS
LIN {X 83.537,Y -43.623,Z -77.706,A -90.000,B 90.000,C 0.000} C_DIS
LIN {X 83.399,Y -43.600,Z -77.533,A -90.000,B 90.000,C 0.000} C_DIS
LIN {X 83.312,Y -43.587,Z -77.419,A -90.000,B 90.000,C 0.000} C_DIS
LIN {X 83.138,Y -43.535,Z -77.167,A -90.000,B 90.000,C 0.000} C_DIS
LIN {X 83.083,Y -43.516,Z -77.085,A -90.000,B 90.000,C 0.000} C_DIS
LIN {X 82.928,Y -43.455,Z -76.888,A -90.000,B 90.000,C 0.000} C_DIS
LIN {X 82.882,Y -43.433,Z -76.826,A -90.000,B 90.000,C 0.000} C_DIS
LIN {X 82.702,Y -43.373,Z -76.599,A -90.000,B 90.000,C 0.000} C_DIS
LIN {X 82.570,Y -43.333,Z -76.415,A -90.000,B 90.000,C 0.000} C_DIS
LIN {X 82.478,Y -43.308,Z -76.282,A -90.000,B 90.000,C 0.000} C_DIS
LIN {X 82.248,Y -43.242,Z -75.937,A -90.000,B 90.000,C 0.000} C_DIS
LIN {X 82.147,Y -43.210,Z -75.777,A -90.000,B 90.000,C 0.000} C_DIS
LIN {X 82.014,Y -43.163,Z -75.551,A -90.000,B 90.000,C 0.000} C_DIS
LIN {X 81.936,Y -43.133,Z -75.411,A -90.000,B 90.000,C 0.000} C_DIS
LIN {X 81.868,Y -43.104,Z -75.278,A -90.000,B 90.000,C 0.000} C_DIS
LIN {X 81.808,Y -43.075,Z -75.154,A -90.000,B 90.000,C 0.000} C_DIS
LIN {X 81.757,Y -43.046,Z -75.036,A -90.000,B 90.000,C 0.000} C_DIS
LIN {X 81.734,Y -43.042,Z -74.980,A -90.000,B 90.000,C 0.000} C_DIS
LIN {X 81.714,Y -43.042,Z -74.926,A -90.000,B 90.000,C 0.000} C_DIS
LIN {X 81.666,Y -43.047,Z -74.775,A -90.000,B 90.000,C 0.000} C_DIS
LIN {X 81.643,Y -43.055,Z -74.684,A -90.000,B 90.000,C 0.000} C_DIS
LIN {X 81.629,Y -43.067,Z -74.599,A -90.000,B 90.000,C 0.000} C_DIS
LIN {X 81.625,Y -43.075,Z -74.560,A -90.000,B 90.000,C 0.000} C_DIS
LIN {X 81.622,Y -43.093,Z -74.485,A -90.000,B 90.000,C 0.000} C_DIS
LIN {X 81.626,Y -43.116,Z -74.418,A -90.000,B 90.000,C 0.000} C_DIS
LIN {X 81.631,Y -43.130,Z -74.387,A -90.000,B 90.000,C 0.000} C_DIS
LIN {X 81.647,Y -43.160,Z -74.329,A -90.000,B 90.000,C 0.000} C_DIS
LIN {X 81.657,Y -43.176,Z -74.303,A -90.000,B 90.000,C 0.000} C_DIS
LIN {X 81.683,Y -43.213,Z -74.255,A -90.000,B 90.000,C 0.000} C_DIS
LIN {X 81.699,Y -43.232,Z -74.234,A -90.000,B 90.000,C 0.000} C_DIS
LIN {X 81.735,Y -43.275,Z -74.196,A -90.000,B 90.000,C 0.000} C_DIS
LIN {X 81.755,Y -43.297,Z -74.179,A -90.000,B 90.000,C 0.000} C_DIS
LIN {X 81.801,Y -43.345,Z -74.150,A -90.000,B 90.000,C 0.000} C_DIS
LIN {X 81.853,Y -43.395,Z -74.127,A -90.000,B 90.000,C 0.000} C_DIS
LIN {X 81.912,Y -43.448,Z -74.110,A -90.000,B 90.000,C 0.000} C_DIS
LIN {X 81.976,Y -43.502,Z -74.098,A -90.000,B 90.000,C 0.000} C_DIS
LIN {X 82.046,Y -43.558,Z -74.092,A -90.000,B 90.000,C 0.000} C_DIS
LIN {X 82.122,Y -43.616,Z -74.092,A -90.000,B 90.000,C 0.000} C_DIS
LIN {X 82.203,Y -43.675,Z -74.098,A -90.000,B 90.000,C 0.000} C_DIS
LIN {X 82.335,Y -43.769,Z -74.115,A -90.000,B 90.000,C 0.000} C_DIS
LIN {X 82.429,Y -43.833,Z -74.134,A -90.000,B 90.000,C 0.000} C_DIS
LIN {X 82.528,Y -43.897,Z -74.157,A -90.000,B 90.000,C 0.000} C_DIS
LIN {X 82.740,Y -44.030,Z -74.219,A -90.000,B 90.000,C 0.000} C_DIS
LIN {X 82.970,Y -44.170,Z -74.299,A -90.000,B 90.000,C 0.000} C_DIS
LIN {X 83.091,Y -44.237,Z -74.346,A -90.000,B 90.000,C 0.000} C_DIS
LIN {X 83.215,Y -44.300,Z -74.397,A -90.000,B 90.000,C 0.000} C_DIS
LIN {X 83.344,Y -44.358,Z -74.453,A -90.000,B 90.000,C 0.000} C_DIS
LIN {X 83.476,Y -44.412,Z -74.513,A -90.000,B 90.000,C 0.000} C_DIS
LIN {X 83.612,Y -44.460,Z -74.576,A -90.000,B 90.000,C 0.000} C_DIS
LIN {X 83.751,Y -44.508,Z -74.644,A -90.000,B 90.000,C 0.000} C_DIS
LIN {X 84.038,Y -44.615,Z -74.791,A -90.000,B 90.000,C 0.000} C_DIS
LIN {X 84.335,Y -44.722,Z -74.952,A -90.000,B 90.000,C 0.000} C_DIS
LIN {X 84.488,Y -44.771,Z -75.037,A -90.000,B 90.000,C 0.000} C_DIS
LIN {X 84.643,Y -44.811,Z -75.126,A -90.000,B 90.000,C 0.000} C_DIS
LIN {X 84.800,Y -44.844,Z -75.218,A -90.000,B 90.000,C 0.000} C_DIS
LIN {X 84.958,Y -44.871,Z -75.313,A -90.000,B 90.000,C 0.000} C_DIS
LIN {X 85.281,Y -44.935,Z -75.512,A -90.000,B 90.000,C 0.000} C_DIS
LIN {X 85.609,Y -44.999,Z -75.721,A -90.000,B 90.000,C 0.000} C_DIS
LIN {X 85.775,Y -45.026,Z -75.830,A -90.000,B 90.000,C 0.000} C_DIS
LIN {X 85.942,Y -45.043,Z -75.940,A -90.000,B 90.000,C 0.000} C_DIS
LIN {X 86.109,Y -45.056,Z -76.053,A -90.000,B 90.000,C 0.000} C_DIS
LIN {X 86.615,Y -45.090,Z -76.405,A -90.000,B 90.000,C 0.000} C_DIS
LIN {X 86.783,Y -45.100,Z -76.526,A -90.000,B 90.000,C 0.000} C_DIS
LIN {X 86.952,Y -45.105,Z -76.648,A -90.000,B 90.000,C 0.000} C_DIS
LIN {X 87.121,Y -45.104,Z -76.772,A -90.000,B 90.000,C 0.000} C_DIS
LIN {X 87.456,Y -45.087,Z -77.025,A -90.000,B 90.000,C 0.000} C_DIS
LIN {X 87.789,Y -45.066,Z -77.282,A -90.000,B 90.000,C 0.000} C_DIS
LIN {X 88.117,Y -45.043,Z -77.543,A -90.000,B 90.000,C 0.000} C_DIS
LIN {X 88.279,Y -45.023,Z -77.675,A -90.000,B 90.000,C 0.000} C_DIS
LIN {X 88.599,Y -44.966,Z -77.941,A -90.000,B 90.000,C 0.000} C_DIS
LIN {X 88.910,Y -44.907,Z -78.208,A -90.000,B 90.000,C 0.000} C_DIS
LIN {X 89.213,Y -44.846,Z -78.476,A -90.000,B 90.000,C 0.000} C_DIS
LIN {X 89.361,Y -44.813,Z -78.611,A -90.000,B 90.000,C 0.000} C_DIS
LIN {X 89.506,Y -44.773,Z -78.745,A -90.000,B 90.000,C 0.000} C_DIS
LIN {X 89.648,Y -44.727,Z -78.878,A -90.000,B 90.000,C 0.000} C_DIS
LIN {X 90.055,Y -44.593,Z -79.277,A -90.000,B 90.000,C 0.000} C_DIS
LIN {X 90.308,Y -44.505,Z -79.540,A -90.000,B 90.000,C 0.000} C_DIS
LIN {X 90.430,Y -44.462,Z -79.670,A -90.000,B 90.000,C 0.000} C_DIS
LIN {X 90.547,Y -44.414,Z -79.799,A -90.000,B 90.000,C 0.000} C_DIS
LIN {X 90.659,Y -44.362,Z -79.927,A -90.000,B 90.000,C 0.000} C_DIS
LIN {X 90.872,Y -44.259,Z -80.179,A -90.000,B 90.000,C 0.000} C_DIS
LIN {X 91.065,Y -44.157,Z -80.425,A -90.000,B 90.000,C 0.000} C_DIS
LIN {X 91.238,Y -44.058,Z -80.664,A -90.000,B 90.000,C 0.000} C_DIS
LIN {X 91.317,Y -44.010,Z -80.781,A -90.000,B 90.000,C 0.000} C_DIS
LIN {X 91.457,Y -43.918,Z -81.009,A -90.000,B 90.000,C 0.000} C_DIS
LIN {X 91.519,Y -43.872,Z -81.119,A -90.000,B 90.000,C 0.000} C_DIS
LIN {X 91.574,Y -43.826,Z -81.227,A -90.000,B 90.000,C 0.000} C_DIS
LIN {X 91.623,Y -43.778,Z -81.333,A -90.000,B 90.000,C 0.000} C_DIS
LIN {X 91.685,Y -43.704,Z -81.486,A -90.000,B 90.000,C 0.000} C_DIS
LIN {X 91.732,Y -43.635,Z -81.633,A -90.000,B 90.000,C 0.000} C_DIS
LIN {X 91.755,Y -43.591,Z -81.728,A -90.000,B 90.000,C 0.000} C_DIS
LIN {X 91.770,Y -43.549,Z -81.819,A -90.000,B 90.000,C 0.000} C_DIS
LIN {X 91.779,Y -43.509,Z -81.907,A -90.000,B 90.000,C 0.000} C_DIS
LIN {X 91.780,Y -43.472,Z -81.993,A -90.000,B 90.000,C 0.000} C_DIS
LIN {X 91.773,Y -43.437,Z -82.074,A -90.000,B 90.000,C 0.000} C_DIS
LIN {X 91.759,Y -43.404,Z -82.152,A -90.000,B 90.000,C 0.000} C_DIS
LIN {X 91.737,Y -43.374,Z -82.227,A -90.000,B 90.000,C 0.000} C_DIS
LIN {X 91.707,Y -43.346,Z -82.298,A -90.000,B 90.000,C 0.000} C_DIS
LIN {X 91.668,Y -43.321,Z -82.365,A -90.000,B 90.000,C 0.000} C_DIS
LIN {X 91.622,Y -43.299,Z -82.428,A -90.000,B 90.000,C 0.000} C_DIS
LIN {X 91.566,Y -43.279,Z -82.487,A -90.000,B 90.000,C 0.000} C_DIS
LIN {X 91.503,Y -43.262,Z -82.542,A -90.000,B 90.000,C 0.000} C_DIS
LIN {X 91.430,Y -43.248,Z -82.592,A -90.000,B 90.000,C 0.000} C_DIS
LIN {X 91.348,Y -43.236,Z -82.639,A -90.000,B 90.000,C 0.000} C_DIS
LIN {X 91.257,Y -43.228,Z -82.680,A -90.000,B 90.000,C 0.000} C_DIS
LIN {X 91.156,Y -43.223,Z -82.717,A -90.000,B 90.000,C 0.000} C_DIS
LIN {X 91.046,Y -43.222,Z -82.750,A -90.000,B 90.000,C 0.000} C_DIS
LIN {X 90.927,Y -43.222,Z -82.777,A -90.000,B 90.000,C 0.000} C_DIS
LIN {X 90.797,Y -43.223,Z -82.800,A -90.000,B 90.000,C 0.000} C_DIS
LIN {X 90.658,Y -43.225,Z -82.817,A -90.000,B 90.000,C 0.000} C_DIS
LIN {X 90.508,Y -43.230,Z -82.830,A -90.000,B 90.000,C 0.000} C_DIS
LIN {X 90.348,Y -43.238,Z -82.837,A -90.000,B 90.000,C 0.000} C_DIS
LIN {X 90.177,Y -43.249,Z -82.838,A -90.000,B 90.000,C 0.000} C_DIS
LIN {X 89.996,Y -43.261,Z -82.834,A -90.000,B 90.000,C 0.000} C_DIS
LIN {X 89.804,Y -43.276,Z -82.825,A -90.000,B 90.000,C 0.000} C_DIS
LIN {X 89.495,Y -43.302,Z -82.800,A -90.000,B 90.000,C 0.000} C_DIS
LIN {X 89.386,Y -43.308,Z -82.788,A -90.000,B 90.000,C 0.000} C_DIS
LIN {X 89.230,Y -43.324,Z -82.771,A -90.000,B 90.000,C 0.000} C_DIS
LIN {X 89.116,Y -43.336,Z -82.756,A -90.000,B 90.000,C 0.000} C_DIS
LIN {X 88.858,Y -43.353,Z -82.712,A -90.000,B 90.000,C 0.000} C_DIS
LIN {X 88.052,Y -43.426,Z -82.576,A -90.000,B 90.000,C 0.000} C_DIS
LIN {X 87.979,Y -43.432,Z -82.562,A -90.000,B 90.000,C 0.000} C_DIS
LIN {X 87.714,Y -43.450,Z -82.503,A -90.000,B 90.000,C 0.000} C_DIS
LIN {X 87.629,Y -43.454,Z -82.483,A -90.000,B 90.000,C 0.000} C_DIS
LIN {X 87.213,Y -43.464,Z -82.382,A -90.000,B 90.000,C 0.000} C_DIS
LIN {X 86.989,Y -43.472,Z -82.318,A -90.000,B 90.000,C 0.000} C_DIS
LIN {X 86.865,Y -43.481,Z -82.281,A -90.000,B 90.000,C 0.000} C_DIS
LIN {X 86.658,Y -43.498,Z -82.212,A -90.000,B 90.000,C 0.000} C_DIS
LIN {X 86.432,Y -43.508,Z -82.129,A -90.000,B 90.000,C 0.000} C_DIS
LIN {X 86.227,Y -43.507,Z -82.047,A -90.000,B 90.000,C 0.000} C_DIS
LIN {X 85.986,Y -43.495,Z -81.937,A -90.000,B 90.000,C 0.000} C_DIS
LIN {X 85.713,Y -43.477,Z -81.808,A -90.000,B 90.000,C 0.000} C_DIS
LIN {X 85.493,Y -43.464,Z -81.700,A -90.000,B 90.000,C 0.000} C_DIS
LIN {X 85.232,Y -43.455,Z -81.557,A -90.000,B 90.000,C 0.000} C_DIS
LIN {X 85.161,Y -43.451,Z -81.515,A -90.000,B 90.000,C 0.000} C_DIS
LIN {X 85.001,Y -43.436,Z -81.421,A -90.000,B 90.000,C 0.000} C_DIS
LIN {X 84.697,Y -43.394,Z -81.236,A -90.000,B 90.000,C 0.000} C_DIS
LIN {X 84.519,Y -43.360,Z -81.118,A -90.000,B 90.000,C 0.000} C_DIS
LIN {X 84.292,Y -43.308,Z -80.959,A -90.000,B 90.000,C 0.000} C_DIS
LIN {X 84.292,Y -43.308,Z -80.958,A -90.000,B 90.000,C 0.000} C_DIS
LIN {X 84.119,Y -43.308,Z -80.564,A -90.000,B 90.000,C 0.000} C_DIS
LIN {X 83.769,Y -43.308,Z -79.952,A -90.000,B 90.000,C 0.000} C_DIS
LIN {X 83.651,Y -43.308,Z -79.655,A -90.000,B 90.000,C 0.000} C_DIS
LIN {X 83.607,Y -43.308,Z -79.512,A -90.000,B 90.000,C 0.000} C_DIS
LIN {X 83.460,Y -43.308,Z -79.035,A -90.000,B 90.000,C 0.000} C_DIS
LIN {X 83.431,Y -43.308,Z -78.912,A -90.000,B 90.000,C 0.000} C_DIS
LIN {X 83.221,Y -43.308,Z -78.343,A -90.000,B 90.000,C 0.000} C_DIS
LIN {X 83.096,Y -43.308,Z -78.105,A -90.000,B 90.000,C 0.000} C_DIS
LIN {X 82.978,Y -43.308,Z -77.774,A -90.000,B 90.000,C 0.000} C_DIS
LIN {X 82.814,Y -43.308,Z -77.249,A -90.000,B 90.000,C 0.000} C_DIS
LIN {X 82.743,Y -43.308,Z -76.951,A -90.000,B 90.000,C 0.000} C_DIS
LIN {X 82.531,Y -43.308,Z -76.416,A -90.000,B 90.000,C 0.000} C_DIS
LIN {X 82.494,Y -43.308,Z -76.318,A -90.000,B 90.000,C 0.000} C_DIS
LIN {X 82.470,Y -43.308,Z -76.264,A -90.000,B 90.000,C 0.000} C_DIS
LIN {X 82.339,Y -43.308,Z -75.909,A -90.000,B 90.000,C 0.000} C_DIS
LIN {X 82.150,Y -43.308,Z -75.218,A -90.000,B 90.000,C 0.000} C_DIS
LIN {X 82.079,Y -43.308,Z -74.953,A -90.000,B 90.000,C 0.000} C_DIS
LIN {X 82.034,Y -43.308,Z -74.844,A -90.000,B 90.000,C 0.000} C_DIS
LIN {X 81.742,Y -43.308,Z -74.099,A -90.000,B 90.000,C 0.000} C_DIS
LIN {X 81.650,Y -43.308,Z -73.767,A -90.000,B 90.000,C 0.000} C_DIS
LIN {X 81.428,Y -43.308,Z -72.901,A -90.000,B 90.000,C 0.000} C_DIS
LIN {X 81.365,Y -43.308,Z -72.736,A -90.000,B 90.000,C 0.000} C_DIS
LIN {X 81.147,Y -43.308,Z -72.066,A -90.000,B 90.000,C 0.000} C_DIS
LIN {X 81.054,Y -43.308,Z -71.653,A -90.000,B 90.000,C 0.000} C_DIS
LIN {X 80.928,Y -43.308,Z -71.018,A -90.000,B 90.000,C 0.000} C_DIS
LIN {X 80.833,Y -43.308,Z -70.420,A -90.000,B 90.000,C 0.000} C_DIS
LIN {X 80.717,Y -43.308,Z -69.811,A -90.000,B 90.000,C 0.000} C_DIS
LIN {X 80.678,Y -43.308,Z -69.372,A -90.000,B 90.000,C 0.000} C_DIS
LIN {X 80.633,Y -43.308,Z -68.813,A -90.000,B 90.000,C 0.000} C_DIS
LIN {X 80.641,Y -43.308,Z -68.027,A -90.000,B 90.000,C 0.000} C_DIS
LIN {X 80.668,Y -43.308,Z -67.734,A -90.000,B 90.000,C 0.000} C_DIS
LIN {X 80.701,Y -43.308,Z -67.430,A -90.000,B 90.000,C 0.000} C_DIS
LIN {X 80.801,Y -43.308,Z -66.461,A -90.000,B 90.000,C 0.000} C_DIS
LIN {X 80.963,Y -43.308,Z -65.604,A -90.000,B 90.000,C 0.000} C_DIS
LIN {X 81.060,Y -43.308,Z -65.229,A -90.000,B 90.000,C 0.000} C_DIS
LIN {X 81.131,Y -43.308,Z -64.973,A -90.000,B 90.000,C 0.000} C_DIS
LIN {X 81.201,Y -43.308,Z -64.741,A -90.000,B 90.000,C 0.000} C_DIS
LIN {X 81.284,Y -43.308,Z -64.519,A -90.000,B 90.000,C 0.000} C_DIS
LIN {X 81.357,Y -43.308,Z -64.338,A -90.000,B 90.000,C 0.000} C_DIS
LIN {X 81.543,Y -43.308,Z -63.893,A -90.000,B 90.000,C 0.000} C_DIS
LIN {X 81.903,Y -43.308,Z -63.152,A -90.000,B 90.000,C 0.000} C_DIS
LIN {X 82.235,Y -43.308,Z -62.569,A -90.000,B 90.000,C 0.000} C_DIS
LIN {X 82.565,Y -43.308,Z -62.001,A -90.000,B 90.000,C 0.000} C_DIS
LIN {X 82.706,Y -43.308,Z -61.763,A -90.000,B 90.000,C 0.000} C_DIS
LIN {X 82.952,Y -43.308,Z -61.402,A -90.000,B 90.000,C 0.000} C_DIS
LIN {X 83.871,Y -43.308,Z -60.140,A -90.000,B 90.000,C 0.000} C_DIS
LIN {X 83.910,Y -43.308,Z -60.087,A -90.000,B 90.000,C 0.000} C_DIS
LIN {X 84.243,Y -43.308,Z -59.630,A -90.000,B 90.000,C 0.000} C_DIS
LIN {X 85.716,Y -43.308,Z -57.875,A -90.000,B 90.000,C 0.000} C_DIS
LIN {X 86.054,Y -43.308,Z -57.499,A -90.000,B 90.000,C 0.000} C_DIS
LIN {X 87.795,Y -43.308,Z -55.685,A -90.000,B 90.000,C 0.000} C_DIS
LIN {X 89.717,Y -43.308,Z -53.926,A -90.000,B 90.000,C 0.000} C_DIS
LIN {X 90.141,Y -43.308,Z -53.541,A -90.000,B 90.000,C 0.000} C_DIS
LIN {X 92.131,Y -43.308,Z -51.836,A -90.000,B 90.000,C 0.000} C_DIS
LIN {X 94.367,Y -43.308,Z -49.945,A -90.000,B 90.000,C 0.000} C_DIS
LIN {X 96.057,Y -43.308,Z -48.464,A -90.000,B 90.000,C 0.000} C_DIS
LIN {X 97.648,Y -43.308,Z -46.921,A -90.000,B 90.000,C 0.000} C_DIS
LIN {X 99.048,Y -43.308,Z -45.444,A -90.000,B 90.000,C 0.000} C_DIS
LIN {X 99.996,Y -43.308,Z -44.391,A -90.000,B 90.000,C 0.000} C_DIS
LIN {X 100.579,Y -43.308,Z -43.768,A -90.000,B 90.000,C 0.000} C_DIS
LIN {X 100.695,Y -43.308,Z -43.644,A -90.000,B 90.000,C 0.000} C_DIS
LIN {X 101.356,Y -43.308,Z -43.005,A -90.000,B 90.000,C 0.000} C_DIS
LIN {X 101.706,Y -43.308,Z -42.673,A -90.000,B 90.000,C 0.000} C_DIS
LIN {X 101.866,Y -43.308,Z -42.532,A -90.000,B 90.000,C 0.000} C_DIS
LIN {X 102.362,Y -43.308,Z -42.117,A -90.000,B 90.000,C 0.000} C_DIS
LIN {X 102.731,Y -43.308,Z -41.815,A -90.000,B 90.000,C 0.000} C_DIS
LIN {X 103.250,Y -43.308,Z -41.423,A -90.000,B 90.000,C 0.000} C_DIS
LIN {X 103.737,Y -43.308,Z -41.074,A -90.000,B 90.000,C 0.000} C_DIS
LIN {X 104.721,Y -43.308,Z -40.448,A -90.000,B 90.000,C 0.000} C_DIS
LIN {X 105.001,Y -43.308,Z -40.293,A -90.000,B 90.000,C 0.000} C_DIS
LIN {X 105.661,Y -43.308,Z -39.943,A -90.000,B 90.000,C 0.000} C_DIS
LIN {X 105.786,Y -43.308,Z -39.882,A -90.000,B 90.000,C 0.000} C_DIS
LIN {X 106.036,Y -43.308,Z -39.758,A -90.000,B 90.000,C 0.000} C_DIS
LIN {X 106.507,Y -43.308,Z -39.550,A -90.000,B 90.000,C 0.000} C_DIS
LIN {X 106.943,Y -43.308,Z -39.372,A -90.000,B 90.000,C 0.000} C_DIS
LIN {X 107.337,Y -43.308,Z -39.216,A -90.000,B 90.000,C 0.000} C_DIS
LIN {X 107.600,Y -43.308,Z -39.133,A -90.000,B 90.000,C 0.000} C_DIS
LIN {X 108.152,Y -43.308,Z -38.987,A -90.000,B 90.000,C 0.000} C_DIS
LIN {X 108.544,Y -43.308,Z -38.895,A -90.000,B 90.000,C 0.000} C_DIS
LIN {X 108.817,Y -43.308,Z -38.855,A -90.000,B 90.000,C 0.000} C_DIS
LIN {X 109.059,Y -43.308,Z -38.830,A -90.000,B 90.000,C 0.000} C_DIS
LIN {X 109.209,Y -43.308,Z -38.818,A -90.000,B 90.000,C 0.000} C_DIS
LIN {X 109.623,Y -43.308,Z -38.792,A -90.000,B 90.000,C 0.000} C_DIS
LIN {X 109.873,Y -43.308,Z -38.784,A -90.000,B 90.000,C 0.000} C_DIS
LIN {X 110.341,Y -43.308,Z -38.810,A -90.000,B 90.000,C 0.000} C_DIS
LIN {X 110.714,Y -43.308,Z -38.880,A -90.000,B 90.000,C 0.000} C_DIS
LIN {X 111.096,Y -43.308,Z -38.974,A -90.000,B 90.000,C 0.000} C_DIS
LIN {X 111.174,Y -43.308,Z -38.999,A -90.000,B 90.000,C 0.000} C_DIS
LIN {X 111.431,Y -43.308,Z -39.097,A -90.000,B 90.000,C 0.000} C_DIS
LIN {X 111.527,Y -43.308,Z -39.140,A -90.000,B 90.000,C 0.000} C_DIS
LIN {X 111.834,Y -43.308,Z -39.310,A -90.000,B 90.000,C 0.000} C_DIS
LIN {X 111.963,Y -43.308,Z -39.395,A -90.000,B 90.000,C 0.000} C_DIS
LIN {X 112.328,Y -43.308,Z -39.668,A -90.000,B 90.000,C 0.000} C_DIS
LIN {X 112.576,Y -43.308,Z -39.918,A -90.000,B 90.000,C 0.000} C_DIS
LIN {X 112.785,Y -43.308,Z -40.200,A -90.000,B 90.000,C 0.000} C_DIS
LIN {X 112.817,Y -43.308,Z -40.255,A -90.000,B 90.000,C 0.000} C_DIS
LIN {X 112.931,Y -43.308,Z -40.461,A -90.000,B 90.000,C 0.000} C_DIS
LIN {X 113.038,Y -43.308,Z -40.685,A -90.000,B 90.000,C 0.000} C_DIS
LIN {X 113.113,Y -43.308,Z -40.868,A -90.000,B 90.000,C 0.000} C_DIS
LIN {X 113.160,Y -43.308,Z -40.993,A -90.000,B 90.000,C 0.000} C_DIS
LIN {X 113.184,Y -43.308,Z -41.079,A -90.000,B 90.000,C 0.000} C_DIS
LIN {X 113.259,Y -43.308,Z -41.422,A -90.000,B 90.000,C 0.000} C_DIS
LIN {X 113.270,Y -43.308,Z -41.511,A -90.000,B 90.000,C 0.000} C_DIS
LIN {X 113.295,Y -43.308,Z -41.862,A -90.000,B 90.000,C 0.000} C_DIS
LIN {X 113.301,Y -43.308,Z -42.092,A -90.000,B 90.000,C 0.000} C_DIS
LIN {X 113.300,Y -43.308,Z -42.154,A -90.000,B 90.000,C 0.000} C_DIS
LIN {X 113.266,Y -43.308,Z -42.505,A -90.000,B 90.000,C 0.000} C_DIS
LIN {X 113.211,Y -43.308,Z -42.777,A -90.000,B 90.000,C 0.000} C_DIS
LIN {X 113.127,Y -43.308,Z -43.119,A -90.000,B 90.000,C 0.000} C_DIS
LIN {X 113.076,Y -43.308,Z -43.290,A -90.000,B 90.000,C 0.000} C_DIS
LIN {X 113.039,Y -43.308,Z -43.398,A -90.000,B 90.000,C 0.000} C_DIS
LIN {X 113.002,Y -43.308,Z -43.491,A -90.000,B 90.000,C 0.000} C_DIS
LIN {X 112.824,Y -43.308,Z -43.992,A -90.000,B 90.000,C 0.000} C_DIS
LIN {X 112.764,Y -43.308,Z -44.149,A -90.000,B 90.000,C 0.000} C_DIS
LIN {X 112.662,Y -43.308,Z -44.440,A -90.000,B 90.000,C 0.000} C_DIS
LIN {X 112.608,Y -43.308,Z -44.601,A -90.000,B 90.000,C 0.000} C_DIS
LIN {X 112.540,Y -43.308,Z -44.820,A -90.000,B 90.000,C 0.000} C_DIS
LIN {X 112.519,Y -43.308,Z -44.964,A -90.000,B 90.000,C 0.000} C_DIS
LIN {X 112.485,Y -43.308,Z -45.536,A -90.000,B 90.000,C 0.000} C_DIS
LIN {X 112.481,Y -43.308,Z -45.743,A -90.000,B 90.000,C 0.000} C_DIS
LIN {X 112.497,Y -43.308,Z -46.115,A -90.000,B 90.000,C 0.000} C_DIS
LIN {X 112.491,Y -43.308,Z -46.484,A -90.000,B 90.000,C 0.000} C_DIS
LIN {X 112.499,Y -43.308,Z -46.747,A -90.000,B 90.000,C 0.000} C_DIS
LIN {X 112.493,Y -43.308,Z -46.880,A -90.000,B 90.000,C 0.000} C_DIS
LIN {X 112.455,Y -43.308,Z -47.594,A -90.000,B 90.000,C 0.000} C_DIS
LIN {X 112.410,Y -43.308,Z -48.089,A -90.000,B 90.000,C 0.000} C_DIS
LIN {X 112.385,Y -43.308,Z -48.324,A -90.000,B 90.000,C 0.000} C_DIS
LIN {X 112.328,Y -43.308,Z -48.723,A -90.000,B 90.000,C 0.000} C_DIS
LIN {X 112.238,Y -43.308,Z -49.219,A -90.000,B 90.000,C 0.000} C_DIS
LIN {X 112.144,Y -43.308,Z -49.681,A -90.000,B 90.000,C 0.000} C_DIS
LIN {X 111.989,Y -43.308,Z -50.301,A -90.000,B 90.000,C 0.000} C_DIS
LIN {X 111.898,Y -43.308,Z -50.637,A -90.000,B 90.000,C 0.000} C_DIS
LIN {X 111.670,Y -43.308,Z -51.398,A -90.000,B 90.000,C 0.000} C_DIS
LIN {X 111.596,Y -43.308,Z -51.621,A -90.000,B 90.000,C 0.000} C_DIS
LIN {X 111.453,Y -43.308,Z -52.038,A -90.000,B 90.000,C 0.000} C_DIS
LIN {X 111.198,Y -43.308,Z -52.697,A -90.000,B 90.000,C 0.000} C_DIS
LIN {X 110.830,Y -43.308,Z -53.669,A -90.000,B 90.000,C 0.000} C_DIS
LIN {X 110.269,Y -43.308,Z -55.115,A -90.000,B 90.000,C 0.000} C_DIS
LIN {X 109.599,Y -43.308,Z -56.785,A -90.000,B 90.000,C 0.000} C_DIS
LIN {X 109.264,Y -43.308,Z -57.691,A -90.000,B 90.000,C 0.000} C_DIS
LIN {X 108.886,Y -43.308,Z -58.683,A -90.000,B 90.000,C 0.000} C_DIS
LIN {X 108.439,Y -43.308,Z -59.961,A -90.000,B 90.000,C 0.000} C_DIS
LIN {X 108.161,Y -43.308,Z -60.725,A -90.000,B 90.000,C 0.000} C_DIS
LIN {X 107.705,Y -43.308,Z -62.017,A -90.000,B 90.000,C 0.000} C_DIS
LIN {X 107.352,Y -43.308,Z -62.981,A -90.000,B 90.000,C 0.000} C_DIS
LIN {X 106.646,Y -43.308,Z -64.864,A -90.000,B 90.000,C 0.000} C_DIS
LIN {X 106.501,Y -43.308,Z -65.232,A -90.000,B 90.000,C 0.000} C_DIS
LIN {X 105.893,Y -43.308,Z -66.700,A -90.000,B 90.000,C 0.000} C_DIS
LIN {X 105.528,Y -43.308,Z -67.536,A -90.000,B 90.000,C 0.000} C_DIS
LIN {X 105.083,Y -43.308,Z -68.484,A -90.000,B 90.000,C 0.000} C_DIS
LIN {X 104.894,Y -43.308,Z -68.882,A -90.000,B 90.000,C 0.000} C_DIS
LIN {X 104.207,Y -43.308,Z -70.253,A -90.000,B 90.000,C 0.000} C_DIS
LIN {X 104.031,Y -43.308,Z -70.589,A -90.000,B 90.000,C 0.000} C_DIS
LIN {X 103.819,Y -43.308,Z -70.969,A -90.000,B 90.000,C 0.000} C_DIS
LIN {X 102.989,Y -43.308,Z -72.447,A -90.000,B 90.000,C 0.000} C_DIS
LIN {X 102.813,Y -43.308,Z -72.746,A -90.000,B 90.000,C 0.000} C_DIS
LIN {X 102.180,Y -43.308,Z -73.759,A -90.000,B 90.000,C 0.000} C_DIS
LIN {X 101.500,Y -43.308,Z -74.793,A -90.000,B 90.000,C 0.000} C_DIS
LIN {X 101.183,Y -43.308,Z -75.230,A -90.000,B 90.000,C 0.000} C_DIS
LIN {X 100.943,Y -43.308,Z -75.553,A -90.000,B 90.000,C 0.000} C_DIS
LIN {X 100.120,Y -43.308,Z -76.590,A -90.000,B 90.000,C 0.000} C_DIS
LIN {X 99.841,Y -43.308,Z -76.933,A -90.000,B 90.000,C 0.000} C_DIS
LIN {X 98.356,Y -43.308,Z -78.477,A -90.000,B 90.000,C 0.000} C_DIS
LIN {X 98.081,Y -43.308,Z -78.738,A -90.000,B 90.000,C 0.000} C_DIS
LIN {X 97.084,Y -43.308,Z -79.645,A -90.000,B 90.000,C 0.000} C_DIS
LIN {X 96.676,Y -43.308,Z -79.996,A -90.000,B 90.000,C 0.000} C_DIS
LIN {X 96.316,Y -43.308,Z -80.271,A -90.000,B 90.000,C 0.000} C_DIS
LIN {X 96.030,Y -43.308,Z -80.476,A -90.000,B 90.000,C 0.000} C_DIS
LIN {X 95.220,Y -43.308,Z -80.949,A -90.000,B 90.000,C 0.000} C_DIS
LIN {X 94.880,Y -43.308,Z -81.141,A -90.000,B 90.000,C 0.000} C_DIS
LIN {X 93.261,Y -43.308,Z -81.941,A -90.000,B 90.000,C 0.000} C_DIS
LIN {X 92.963,Y -43.308,Z -82.057,A -90.000,B 90.000,C 0.000} C_DIS
LIN {X 91.280,Y -43.308,Z -82.489,A -90.000,B 90.000,C 0.000} C_DIS
LIN {X 90.968,Y -43.308,Z -82.557,A -90.000,B 90.000,C 0.000} C_DIS
LIN {X 90.773,Y -43.308,Z -82.582,A -90.000,B 90.000,C 0.000} C_DIS
LIN {X 89.754,Y -43.308,Z -82.736,A -90.000,B 90.000,C 0.000} C_DIS
LIN {X 89.081,Y -43.308,Z -82.832,A -90.000,B 90.000,C 0.000} C_DIS
LIN {X 88.931,Y -43.308,Z -82.831,A -90.000,B 90.000,C 0.000} C_DIS
LIN {X 88.563,Y -43.308,Z -82.862,A -90.000,B 90.000,C 0.000} C_DIS
LIN {X 88.219,Y -43.308,Z -82.895,A -90.000,B 90.000,C 0.000} C_DIS
LIN {X 88.097,Y -43.308,Z -82.925,A -90.000,B 90.000,C 0.000} C_DIS
LIN {X 87.818,Y -43.308,Z -82.971,A -90.000,B 90.000,C 0.000} C_DIS
LIN {X 87.428,Y -43.308,Z -82.967,A -90.000,B 90.000,C 0.000} C_DIS
LIN {X 87.107,Y -43.308,Z -82.916,A -90.000,B 90.000,C 0.000} C_DIS
LIN {X 86.396,Y -43.308,Z -82.896,A -90.000,B 90.000,C 0.000} C_DIS
LIN {X 86.163,Y -43.308,Z -82.854,A -90.000,B 90.000,C 0.000} C_DIS
LIN {X 85.945,Y -43.308,Z -82.764,A -90.000,B 90.000,C 0.000} C_DIS
LIN {X 85.749,Y -43.308,Z -82.630,A -90.000,B 90.000,C 0.000} C_DIS
LIN {X 85.606,Y -43.308,Z -82.519,A -90.000,B 90.000,C 0.000} C_DIS
LIN {X 84.992,Y -43.308,Z -82.082,A -90.000,B 90.000,C 0.000} C_DIS
LIN {X 84.829,Y -43.308,Z -81.910,A -90.000,B 90.000,C 0.000} C_DIS
LIN {X 84.589,Y -43.308,Z -81.579,A -90.000,B 90.000,C 0.000} C_DIS
LIN {X 84.456,Y -43.308,Z -81.333,A -90.000,B 90.000,C 0.000} C_DIS
LIN {X 84.292,Y -43.308,Z -80.958,A -90.000,B 90.000,C 0.000} C_DIS
LIN {X 84.292,Y -60.000,Z -80.958,A -90.000,B 90.000,C 0.000} C_DIS
LIN {X 16.580,Y -60.000,Z -126.268,A -90.000,B 90.000,C 0.000} C_DIS
LIN {X 16.580,Y -47.986,Z -126.268,A -90.000,B 90.000,C 0.000} C_DIS
LIN {X 15.723,Y -48.102,Z -127.560,A -90.000,B 90.000,C 0.000} C_DIS
LIN {X 15.614,Y -48.113,Z -127.724,A -90.000,B 90.000,C 0.000} C_DIS
LIN {X 15.426,Y -48.127,Z -127.944,A -90.000,B 90.000,C 0.000} C_DIS
LIN {X 15.145,Y -48.145,Z -128.223,A -90.000,B 90.000,C 0.000} C_DIS
LIN {X 14.200,Y -48.207,Z -129.157,A -90.000,B 90.000,C 0.000} C_DIS
LIN {X 14.098,Y -48.214,Z -129.256,A -90.000,B 90.000,C 0.000} C_DIS
LIN {X 13.743,Y -48.230,Z -129.442,A -90.000,B 90.000,C 0.000} C_DIS
LIN {X 12.339,Y -48.292,Z -130.173,A -90.000,B 90.000,C 0.000} C_DIS
LIN {X 12.107,Y -48.297,Z -130.291,A -90.000,B 90.000,C 0.000} C_DIS
LIN {X 11.925,Y -48.298,Z -130.384,A -90.000,B 90.000,C 0.000} C_DIS
LIN {X 11.787,Y -48.299,Z -130.453,A -90.000,B 90.000,C 0.000} C_DIS
LIN {X 11.581,Y -48.300,Z -130.489,A -90.000,B 90.000,C 0.000} C_DIS
LIN {X 11.107,Y -48.304,Z -130.558,A -90.000,B 90.000,C 0.000} C_DIS
LIN {X 10.082,Y -48.311,Z -130.698,A -90.000,B 90.000,C 0.000} C_DIS
LIN {X 9.808,Y -48.313,Z -130.736,A -90.000,B 90.000,C 0.000} C_DIS
LIN {X 9.605,Y -48.311,Z -130.764,A -90.000,B 90.000,C 0.000} C_DIS
LIN {X 9.240,Y -48.299,Z -130.811,A -90.000,B 90.000,C 0.000} C_DIS
LIN {X 8.565,Y -48.273,Z -130.805,A -90.000,B 90.000,C 0.000} C_DIS
LIN {X 7.293,Y -48.225,Z -130.782,A -90.000,B 90.000,C 0.000} C_DIS
LIN {X 6.932,Y -48.212,Z -130.770,A -90.000,B 90.000,C 0.000} C_DIS
LIN {X 7.686,Y -48.218,Z -130.049,A -90.000,B 90.000,C 0.000} C_DIS
LIN {X 8.011,Y -48.222,Z -129.750,A -90.000,B 90.000,C 0.000} C_DIS
LIN {X 8.708,Y -48.235,Z -129.270,A -90.000,B 90.000,C 0.000} C_DIS
LIN {X 9.584,Y -48.208,Z -128.671,A -90.000,B 90.000,C 0.000} C_DIS
LIN {X 11.986,Y -48.161,Z -127.466,A -90.000,B 90.000,C 0.000} C_DIS
LIN {X 13.559,Y -48.109,Z -126.986,A -90.000,B 90.000,C 0.000} C_DIS
LIN {X 15.597,Y -48.016,Z -126.368,A -90.000,B 90.000,C 0.000} C_DIS
LIN {X 16.580,Y -47.986,Z -126.268,A -90.000,B 90.000,C 0.000} C_DIS
LIN {X 16.516,Y -48.000,Z -126.367,A -90.000,B 90.000,C 0.000} C_DIS
LIN {X 16.455,Y -48.009,Z -126.467,A -90.000,B 90.000,C 0.000} C_DIS
LIN {X 16.338,Y -48.027,Z -126.673,A -90.000,B 90.000,C 0.000} C_DIS
LIN {X 16.230,Y -48.045,Z -126.885,A -90.000,B 90.000,C 0.000} C_DIS
LIN {X 16.130,Y -48.064,Z -127.102,A -90.000,B 90.000,C 0.000} C_DIS
LIN {X 16.082,Y -48.073,Z -127.212,A -90.000,B 90.000,C 0.000} C_DIS
LIN {X 15.993,Y -48.091,Z -127.437,A -90.000,B 90.000,C 0.000} C_DIS
LIN {X 15.910,Y -48.105,Z -127.665,A -90.000,B 90.000,C 0.000} C_DIS
LIN {X 15.830,Y -48.115,Z -127.896,A -90.000,B 90.000,C 0.000} C_DIS
LIN {X 15.725,Y -48.127,Z -128.144,A -90.000,B 90.000,C 0.000} C_DIS
LIN {X 15.637,Y -48.135,Z -128.329,A -90.000,B 90.000,C 0.000} C_DIS
LIN {X 15.490,Y -48.149,Z -128.650,A -90.000,B 90.000,C 0.000} C_DIS
LIN {X 15.395,Y -48.159,Z -128.865,A -90.000,B 90.000,C 0.000} C_DIS
LIN {X 15.212,Y -48.177,Z -129.301,A -90.000,B 90.000,C 0.000} C_DIS
LIN {X 14.989,Y -48.200,Z -129.848,A -90.000,B 90.000,C 0.000} C_DIS
LIN {X 14.650,Y -48.228,Z -130.477,A -90.000,B 90.000,C 0.000} C_DIS
LIN {X 14.479,Y -48.239,Z -130.697,A -90.000,B 90.000,C 0.000} C_DIS
LIN {X 14.344,Y -48.247,Z -130.861,A -90.000,B 90.000,C 0.000} C_DIS
LIN {X 14.135,Y -48.251,Z -131.101,A -90.000,B 90.000,C 0.000} C_DIS
LIN {X 13.914,Y -48.255,Z -131.332,A -90.000,B 90.000,C 0.000} C_DIS
LIN {X 13.679,Y -48.258,Z -131.554,A -90.000,B 90.000,C 0.000} C_DIS
LIN {X 13.514,Y -48.261,Z -131.695,A -90.000,B 90.000,C 0.000} C_DIS
LIN {X 13.428,Y -48.262,Z -131.762,A -90.000,B 90.000,C 0.000} C_DIS
LIN {X 13.251,Y -48.264,Z -131.894,A -90.000,B 90.000,C 0.000} C_DIS
LIN {X 13.159,Y -48.266,Z -131.958,A -90.000,B 90.000,C 0.000} C_DIS
LIN {X 12.968,Y -48.268,Z -132.081,A -90.000,B 90.000,C 0.000} C_DIS
LIN {X 12.869,Y -48.269,Z -132.140,A -90.000,B 90.000,C 0.000} C_DIS
LIN {X 12.664,Y -48.270,Z -132.251,A -90.000,B 90.000,C 0.000} C_DIS
LIN {X 12.515,Y -48.271,Z -132.327,A -90.000,B 90.000,C 0.000} C_DIS
LIN {X 12.439,Y -48.271,Z -132.365,A -90.000,B 90.000,C 0.000} C_DIS
LIN {X 12.406,Y -48.272,Z -132.376,A -90.000,B 90.000,C 0.000} C_DIS
LIN {X 11.864,Y -48.277,Z -132.470,A -90.000,B 90.000,C 0.000} C_DIS
LIN {X 11.378,Y -48.282,Z -132.539,A -90.000,B 90.000,C 0.000} C_DIS
LIN {X 9.870,Y -48.299,Z -132.746,A -90.000,B 90.000,C 0.000} C_DIS
LIN {X 9.359,Y -48.305,Z -132.812,A -90.000,B 90.000,C 0.000} C_DIS
LIN {X 8.853,Y -48.311,Z -132.807,A -90.000,B 90.000,C 0.000} C_DIS
LIN {X 8.538,Y -48.315,Z -132.804,A -90.000,B 90.000,C 0.000} C_DIS
LIN {X 8.307,Y -48.315,Z -132.801,A -90.000,B 90.000,C 0.000} C_DIS
LIN {X 7.208,Y -48.252,Z -132.781,A -90.000,B 90.000,C 0.000} C_DIS
LIN {X 6.546,Y -48.214,Z -132.757,A -90.000,B 90.000,C 0.000} C_DIS
LIN {X 4.923,Y -48.150,Z -132.241,A -90.000,B 90.000,C 0.000} C_DIS
LIN {X 4.668,Y -48.136,Z -132.159,A -90.000,B 90.000,C 0.000} C_DIS
LIN {X 4.621,Y -48.134,Z -132.117,A -90.000,B 90.000,C 0.000} C_DIS
LIN {X 4.423,Y -48.118,Z -131.938,A -90.000,B 90.000,C 0.000} C_DIS
LIN {X 4.215,Y -48.098,Z -131.752,A -90.000,B 90.000,C 0.000} C_DIS
LIN {X 3.951,Y -48.070,Z -131.533,A -90.000,B 90.000,C 0.000} C_DIS
LIN {X 3.953,Y -48.070,Z -131.507,A -90.000,B 90.000,C 0.000} C_DIS
LIN {X 3.973,Y -48.071,Z -131.476,A -90.000,B 90.000,C 0.000} C_DIS
LIN {X 4.093,Y -48.074,Z -131.289,A -90.000,B 90.000,C 0.000} C_DIS
LIN {X 5.026,Y -48.064,Z -129.831,A -90.000,B 90.000,C 0.000} C_DIS
LIN {X 6.334,Y -48.093,Z -128.581,A -90.000,B 90.000,C 0.000} C_DIS
LIN {X 6.574,Y -48.097,Z -128.359,A -90.000,B 90.000,C 0.000} C_DIS
LIN {X 6.765,Y -48.092,Z -128.184,A -90.000,B 90.000,C 0.000} C_DIS
LIN {X 7.402,Y -48.082,Z -127.747,A -90.000,B 90.000,C 0.000} C_DIS
LIN {X 8.567,Y -48.046,Z -126.952,A -90.000,B 90.000,C 0.000} C_DIS
LIN {X 9.069,Y -48.037,Z -126.699,A -90.000,B 90.000,C 0.000} C_DIS
LIN {X 10.821,Y -48.003,Z -125.820,A -90.000,B 90.000,C 0.000} C_DIS
LIN {X 10.956,Y -48.000,Z -125.752,A -90.000,B 90.000,C 0.000} C_DIS
LIN {X 11.240,Y -47.991,Z -125.610,A -90.000,B 90.000,C 0.000} C_DIS
LIN {X 12.213,Y -47.974,Z -125.312,A -90.000,B 90.000,C 0.000} C_DIS
LIN {X 13.185,Y -47.954,Z -125.015,A -90.000,B 90.000,C 0.000} C_DIS
LIN {X 13.644,Y -47.942,Z -124.875,A -90.000,B 90.000,C 0.000} C_DIS
LIN {X 15.197,Y -47.872,Z -124.404,A -90.000,B 90.000,C 0.000} C_DIS
LIN {X 18.430,Y -47.779,Z -124.073,A -90.000,B 90.000,C 0.000} C_DIS
LIN {X 18.593,Y -47.778,Z -124.102,A -90.000,B 90.000,C 0.000} C_DIS
LIN {X 19.517,Y -47.739,Z -124.269,A -90.000,B 90.000,C 0.000} C_DIS
LIN {X 19.531,Y -47.744,Z -124.415,A -90.000,B 90.000,C 0.000} C_DIS
LIN {X 19.448,Y -47.762,Z -124.794,A -90.000,B 90.000,C 0.000} C_DIS
LIN {X 19.363,Y -47.784,Z -125.190,A -90.000,B 90.000,C 0.000} C_DIS
LIN {X 18.606,Y -47.902,Z -126.755,A -90.000,B 90.000,C 0.000} C_DIS
LIN {X 18.510,Y -47.914,Z -126.955,A -90.000,B 90.000,C 0.000} C_DIS
LIN {X 18.452,Y -47.921,Z -127.068,A -90.000,B 90.000,C 0.000} C_DIS
LIN {X 18.392,Y -47.928,Z -127.154,A -90.000,B 90.000,C 0.000} C_DIS
LIN {X 17.698,Y -48.003,Z -128.199,A -90.000,B 90.000,C 0.000} C_DIS
LIN {X 17.211,Y -48.045,Z -128.931,A -90.000,B 90.000,C 0.000} C_DIS
LIN {X 16.893,Y -48.070,Z -129.306,A -90.000,B 90.000,C 0.000} C_DIS
LIN {X 16.476,Y -48.102,Z -129.720,A -90.000,B 90.000,C 0.000} C_DIS
LIN {X 16.216,Y -48.119,Z -129.977,A -90.000,B 90.000,C 0.000} C_DIS
LIN {X 15.492,Y -48.166,Z -130.691,A -90.000,B 90.000,C 0.000} C_DIS
LIN {X 15.254,Y -48.182,Z -130.905,A -90.000,B 90.000,C 0.000} C_DIS
LIN {X 15.008,Y -48.197,Z -131.037,A -90.000,B 90.000,C 0.000} C_DIS
LIN {X 14.336,Y -48.220,Z -131.390,A -90.000,B 90.000,C 0.000} C_DIS
LIN {X 13.252,Y -48.256,Z -131.952,A -90.000,B 90.000,C 0.000} C_DIS
LIN {X 12.829,Y -48.270,Z -132.167,A -90.000,B 90.000,C 0.000} C_DIS
LIN {X 12.664,Y -48.270,Z -132.251,A -90.000,B 90.000,C 0.000} C_DIS
LIN {X 12.576,Y -48.271,Z -132.297,A -90.000,B 90.000,C 0.000} C_DIS
LIN {X 12.448,Y -48.272,Z -132.371,A -90.000,B 90.000,C 0.000} C_DIS
LIN {X 12.414,Y -48.272,Z -132.386,A -90.000,B 90.000,C 0.000} C_DIS
LIN {X 12.310,Y -48.273,Z -132.415,A -90.000,B 90.000,C 0.000} C_DIS
LIN {X 12.128,Y -48.274,Z -132.474,A -90.000,B 90.000,C 0.000} C_DIS
LIN {X 11.951,Y -48.275,Z -132.542,A -90.000,B 90.000,C 0.000} C_DIS
LIN {X 11.691,Y -48.277,Z -132.652,A -90.000,B 90.000,C 0.000} C_DIS
LIN {X 11.439,Y -48.278,Z -132.777,A -90.000,B 90.000,C 0.000} C_DIS
LIN {X 11.194,Y -48.279,Z -132.915,A -90.000,B 90.000,C 0.000} C_DIS
LIN {X 10.954,Y -48.279,Z -133.065,A -90.000,B 90.000,C 0.000} C_DIS
LIN {X 10.642,Y -48.280,Z -133.278,A -90.000,B 90.000,C 0.000} C_DIS
LIN {X 10.488,Y -48.278,Z -133.389,A -90.000,B 90.000,C 0.000} C_DIS
LIN {X 10.335,Y -48.271,Z -133.502,A -90.000,B 90.000,C 0.000} C_DIS
LIN {X 9.878,Y -48.246,Z -133.844,A -90.000,B 90.000,C 0.000} C_DIS
LIN {X 9.417,Y -48.220,Z -134.153,A -90.000,B 90.000,C 0.000} C_DIS
LIN {X 9.222,Y -48.210,Z -134.280,A -90.000,B 90.000,C 0.000} C_DIS
LIN {X 9.023,Y -48.200,Z -134.379,A -90.000,B 90.000,C 0.000} C_DIS
LIN {X 8.779,Y -48.188,Z -134.487,A -90.000,B 90.000,C 0.000} C_DIS
LIN {X 8.614,Y -48.180,Z -134.552,A -90.000,B 90.000,C 0.000} C_DIS
LIN {X 8.445,Y -48.171,Z -134.610,A -90.000,B 90.000,C 0.000} C_DIS
LIN {X 8.359,Y -48.167,Z -134.636,A -90.000,B 90.000,C 0.000} C_DIS
LIN {X 8.185,Y -48.159,Z -134.683,A -90.000,B 90.000,C 0.000} C_DIS
LIN {X 8.007,Y -48.151,Z -134.721,A -90.000,B 90.000,C 0.000} C_DIS
LIN {X 7.916,Y -48.147,Z -134.737,A -90.000,B 90.000,C 0.000} C_DIS
LIN {X 7.731,Y -48.138,Z -134.762,A -90.000,B 90.000,C 0.000} C_DIS
LIN {X 7.542,Y -48.130,Z -134.776,A -90.000,B 90.000,C 0.000} C_DIS
LIN {X 7.347,Y -48.120,Z -134.779,A -90.000,B 90.000,C 0.000} C_DIS
LIN {X 7.152,Y -48.114,Z -134.775,A -90.000,B 90.000,C 0.000} C_DIS
LIN {X 6.831,Y -48.096,Z -134.765,A -90.000,B 90.000,C 0.000} C_DIS
LIN {X 6.182,Y -48.058,Z -134.740,A -90.000,B 90.000,C 0.000} C_DIS
LIN {X 6.015,Y -48.052,Z -134.680,A -90.000,B 90.000,C 0.000} C_DIS
LIN {X 3.832,Y -47.985,Z -133.987,A -90.000,B 90.000,C 0.000} C_DIS
LIN {X 3.661,Y -47.977,Z -133.932,A -90.000,B 90.000,C 0.000} C_DIS
LIN {X 3.494,Y -47.971,Z -133.783,A -90.000,B 90.000,C 0.000} C_DIS
LIN {X 2.982,Y -47.929,Z -133.320,A -90.000,B 90.000,C 0.000} C_DIS
LIN {X 2.919,Y -47.923,Z -133.266,A -90.000,B 90.000,C 0.000} C_DIS
LIN {X 1.960,Y -47.840,Z -132.471,A -90.000,B 90.000,C 0.000} C_DIS
LIN {X 1.893,Y -47.836,Z -132.345,A -90.000,B 90.000,C 0.000} C_DIS
LIN {X 1.987,Y -47.875,Z -131.134,A -90.000,B 90.000,C 0.000} C_DIS
LIN {X 1.998,Y -47.877,Z -130.992,A -90.000,B 90.000,C 0.000} C_DIS
LIN {X 2.010,Y -47.875,Z -130.851,A -90.000,B 90.000,C 0.000} C_DIS
LIN {X 2.131,Y -47.878,Z -130.662,A -90.000,B 90.000,C 0.000} C_DIS
LIN {X 3.447,Y -47.867,Z -128.607,A -90.000,B 90.000,C 0.000} C_DIS
LIN {X 3.518,Y -47.868,Z -128.520,A -90.000,B 90.000,C 0.000} C_DIS
LIN {X 4.239,Y -47.886,Z -127.829,A -90.000,B 90.000,C 0.000} C_DIS
LIN {X 4.425,Y -47.887,Z -127.651,A -90.000,B 90.000,C 0.000} C_DIS
LIN {X 4.991,Y -47.870,Z -127.115,A -90.000,B 90.000,C 0.000} C_DIS
LIN {X 5.525,Y -47.855,Z -126.628,A -90.000,B 90.000,C 0.000} C_DIS
LIN {X 6.307,Y -47.851,Z -126.089,A -90.000,B 90.000,C 0.000} C_DIS
LIN {X 7.551,Y -47.832,Z -125.237,A -90.000,B 90.000,C 0.000} C_DIS
LIN {X 8.173,Y -47.834,Z -124.923,A -90.000,B 90.000,C 0.000} C_DIS
LIN {X 9.017,Y -47.827,Z -124.498,A -90.000,B 90.000,C 0.000} C_DIS
LIN {X 10.061,Y -47.805,Z -123.974,A -90.000,B 90.000,C 0.000} C_DIS
LIN {X 10.495,Y -47.791,Z -123.757,A -90.000,B 90.000,C 0.000} C_DIS
LIN {X 11.628,Y -47.772,Z -123.411,A -90.000,B 90.000,C 0.000} C_DIS
LIN {X 14.797,Y -47.706,Z -122.442,A -90.000,B 90.000,C 0.000} C_DIS
LIN {X 15.118,Y -47.706,Z -122.408,A -90.000,B 90.000,C 0.000} C_DIS
LIN {X 15.424,Y -47.704,Z -122.377,A -90.000,B 90.000,C 0.000} C_DIS
LIN {X 18.502,Y -47.622,Z -122.061,A -90.000,B 90.000,C 0.000} C_DIS
LIN {X 19.954,Y -47.613,Z -122.319,A -90.000,B 90.000,C 0.000} C_DIS
LIN {X 20.941,Y -47.573,Z -122.497,A -90.000,B 90.000,C 0.000} C_DIS
LIN {X 21.162,Y -47.571,Z -122.669,A -90.000,B 90.000,C 0.000} C_DIS
LIN {X 21.467,Y -47.569,Z -122.907,A -90.000,B 90.000,C 0.000} C_DIS
LIN {X 21.463,Y -47.571,Z -122.956,A -90.000,B 90.000,C 0.000} C_DIS
LIN {X 21.453,Y -47.592,Z -123.334,A -90.000,B 90.000,C 0.000} C_DIS
LIN {X 21.452,Y -47.597,Z -123.426,A -90.000,B 90.000,C 0.000} C_DIS
LIN {X 21.460,Y -47.604,Z -123.567,A -90.000,B 90.000,C 0.000} C_DIS
LIN {X 21.546,Y -47.636,Z -124.547,A -90.000,B 90.000,C 0.000} C_DIS
LIN {X 21.400,Y -47.669,Z -125.222,A -90.000,B 90.000,C 0.000} C_DIS
LIN {X 21.264,Y -47.701,Z -125.850,A -90.000,B 90.000,C 0.000} C_DIS
LIN {X 21.012,Y -47.732,Z -126.370,A -90.000,B 90.000,C 0.000} C_DIS
LIN {X 20.302,Y -47.813,Z -127.837,A -90.000,B 90.000,C 0.000} C_DIS
LIN {X 20.167,Y -47.828,Z -128.101,A -90.000,B 90.000,C 0.000} C_DIS
LIN {X 20.029,Y -47.842,Z -128.300,A -90.000,B 90.000,C 0.000} C_DIS
LIN {X 19.683,Y -47.876,Z -128.822,A -90.000,B 90.000,C 0.000} C_DIS
LIN {X 18.809,Y -47.924,Z -130.133,A -90.000,B 90.000,C 0.000} C_DIS
LIN {X 18.356,Y -47.955,Z -130.667,A -90.000,B 90.000,C 0.000} C_DIS
LIN {X 17.584,Y -48.012,Z -131.433,A -90.000,B 90.000,C 0.000} C_DIS
LIN {X 17.308,Y -48.029,Z -131.706,A -90.000,B 90.000,C 0.000} C_DIS
LIN {X 17.196,Y -48.032,Z -131.816,A -90.000,B 90.000,C 0.000} C_DIS
LIN {X 16.855,Y -48.033,Z -132.149,A -90.000,B 90.000,C 0.000} C_DIS
LIN {X 16.399,Y -48.035,Z -132.557,A -90.000,B 90.000,C 0.000} C_DIS
LIN {X 16.299,Y -48.038,Z -132.609,A -90.000,B 90.000,C 0.000} C_DIS
LIN {X 16.020,Y -48.046,Z -132.758,A -90.000,B 90.000,C 0.000} C_DIS
LIN {X 15.251,Y -48.068,Z -133.162,A -90.000,B 90.000,C 0.000} C_DIS
LIN {X 14.184,Y -48.100,Z -133.715,A -90.000,B 90.000,C 0.000} C_DIS
LIN {X 13.209,Y -48.128,Z -134.211,A -90.000,B 90.000,C 0.000} C_DIS
LIN {X 13.036,Y -48.131,Z -134.269,A -90.000,B 90.000,C 0.000} C_DIS
LIN {X 12.883,Y -48.130,Z -134.320,A -90.000,B 90.000,C 0.000} C_DIS
LIN {X 12.172,Y -48.146,Z -134.442,A -90.000,B 90.000,C 0.000} C_DIS
LIN {X 11.649,Y -48.160,Z -134.517,A -90.000,B 90.000,C 0.000} C_DIS
LIN {X 11.505,Y -48.161,Z -134.537,A -90.000,B 90.000,C 0.000} C_DIS
LIN {X 10.115,Y -48.143,Z -134.725,A -90.000,B 90.000,C 0.000} C_DIS
LIN {X 9.475,Y -48.131,Z -134.806,A -90.000,B 90.000,C 0.000} C_DIS
LIN {X 8.566,Y -48.127,Z -134.796,A -90.000,B 90.000,C 0.000} C_DIS
LIN {X 7.360,Y -48.121,Z -134.779,A -90.000,B 90.000,C 0.000} C_DIS
LIN {X 7.347,Y -48.120,Z -134.779,A -90.000,B 90.000,C 0.000} C_DIS
LIN {X 7.229,Y -48.122,Z -134.778,A -90.000,B 90.000,C 0.000} C_DIS
LIN {X 7.111,Y -48.117,Z -134.779,A -90.000,B 90.000,C 0.000} C_DIS
LIN {X 6.993,Y -48.110,Z -134.783,A -90.000,B 90.000,C 0.000} C_DIS
LIN {X 6.756,Y -48.097,Z -134.796,A -90.000,B 90.000,C 0.000} C_DIS
LIN {X 6.519,Y -48.083,Z -134.819,A -90.000,B 90.000,C 0.000} C_DIS
LIN {X 6.179,Y -48.064,Z -134.867,A -90.000,B 90.000,C 0.000} C_DIS
LIN {X 5.996,Y -48.054,Z -134.849,A -90.000,B 90.000,C 0.000} C_DIS
LIN {X 5.599,Y -48.032,Z -134.838,A -90.000,B 90.000,C 0.000} C_DIS
LIN {X 5.372,Y -48.019,Z -134.838,A -90.000,B 90.000,C 0.000} C_DIS
LIN {X 5.031,Y -48.000,Z -134.850,A -90.000,B 90.000,C 0.000} C_DIS
LIN {X 4.804,Y -47.987,Z -134.864,A -90.000,B 90.000,C 0.000} C_DIS
